(* Logix 5000 project; controller R5_CSS vendor 1 type 14 code 74 rev 19.11; software revision 19.01; part 2 of 20 *)
(* tags used below, declared in another part *)
   AC102A : ANALYTICAL;   // QUENCH WATER CONDUCTIVITY CONTROL
   AlarmMaster : DINT;
   AlarmMasterDisable : BOOL;
   FC101 : FLOW_CONTROL;   // QUENCH BASIN FLOW TRANSMITTER CONTROL
   FC108 : FLOW_CONTROL;   // QUENCH FEED FLOW TRANSMITTER
   FC140A : FLOW_CONTROL;   // QUENCH TOWER UPPER SPRAY FLOW CONTROL
   FC140B : FLOW_CONTROL;   // QUENCH TOWER LOWER SPRAY FLOW CONTROL
   FC215 : FLOW_CONTROL;   // OVERHEAD CONDENSER CHILLED WATER FLOW CONTROL
   FC365 : FLOW_CONTROL;   // COALESCER PROCESS IMPURITY FLOW CONTROL
   FC370 : FLOW_CONTROL;   // COALESCER MAKE UP WATER FLOW CONTROL
   FC403 : FLOW_CONTROL;   // COALESCER FLOW CONTROLLER FEEDS TCV108
   FC406 : FLOW_CONTROL;   // HX COOLING WATER FLOW CONTROL
   LC101 : LEVEL_CONTROL;   // QUENCH TOWER BASIN LIT
   LC205 : LEVEL_CONTROL;   // OVERHEAD CONDENSER BASIN LEVEL CONTROL
   LC302 : LEVEL_CONTROL;   // COALESCER OIL CHAMBER LEVEL CONTROL
   LC304 : LEVEL_CONTROL;   // SETTLER SECONDARY TANK INTERFACE LEVEL
   Major : DINT;
   Minor : DINT;
   My_Gateway : DINT[4];
   My_IP_Address : DINT[4];
   My_Subnet : DINT[4];
   MyDint : DINT;
   P101A : PUMP_CONTROL;
   P101B : PUMP_CONTROL;
   P302A : PUMP_CONTROL;
   P303A : PUMP_CONTROL;
   P303B : PUMP_CONTROL;
   PC101A : PRESSURE_CONTROL;   // LOWER QUENCH TOWER PRESSURE TRANSMITTER
   PC101B : PRESSURE_CONTROL;   // UPPER QUENCH TOWER PRESSURE TRANSMITTER PRESSURE CONTOL
   PC102A : PRESSURE_CONTROL;   // QUENCH BASIN TRANSFER PUMP SUCTION PRESSURE CONTROL
   PC102B : PRESSURE_CONTROL;   // QUENCH BASIN TRANSFER PUMP DISCHARGE PRESSURE CONTROL
   PC132 : PRESSURE_CONTROL;
   PC133 : PRESSURE_CONTROL;
   PC134 : PRESSURE_CONTROL;
   PC214 : PRESSURE_CONTROL;   // VACUUM SYSTEM PRESSURE TRANSMITTER
   PC271 : PRESSURE_CONTROL;   // VENT HEADER PRESSURE CONTROL
   PC407A : PRESSURE_CONTROL;   // PRE HX LOW PRESSURE TRANSMITTER
   PC407B : PRESSURE_CONTROL;   // POST HX LOW PRESSURE TRANSMITTER
   PC408 : PRESSURE_CONTROL;

   PID_JHE102_TON : TIMER := (PRE := 500, ACC := 144, EN := 1, TT := 1);
   PID_JHE114B : PID := (CTL := 4864, OLH := 1, DVPA := 1, PVLA := 1, SP := 130.0, KP := 10.0, KI := 5.0, MAXS := 4095.0, SO := 50.0, MAXO := 50.0, UPD := 1.0, PV := -75.0, ERR := 205.0, OUT := 50.0, MAXI := 4095.0, MAXCV := 100.0, MAXTIE := 4095.0, DATA[0] := 0.009664765, DATA[1] := 29.30403, DATA[2] := -75.0, DATA[3] := 205.0, DATA[4] := 130.0, DATA[5] := 0.024420025, DATA[6] := 1.0, DATA[7] := 16.0, DATA[8] := 10.0, DATA[9] := 5.0, DATA[11] := 10.0, DATA[12] := 5.0, DATA[15] := 1.0, DATA[16] := 0.024420025);
   PID_JHE114B_TON : TIMER := (PRE := 500);
   PID_JHE313A : PID := (CTL := 4231808, NDF := 1, INI := 1, OLH := 1, DVPA := 1, PVHA := 1, SP := 135.0, KP := 10.0, KI := 5.0, MAXS := 200.0, SO := 50.0, MAXO := 50.0, UPD := 1.0, PV := 59.625, ERR := 75.375, OUT := 50.0, MAXI := 200.0, MAXCV := 100.0, MAXTIE := 4095.0, DATA[0] := -484.5469, DATA[1] := -477.0, DATA[2] := 59.625, DATA[3] := 75.375, DATA[4] := 135.0, DATA[5] := 0.5, DATA[6] := 1.0, DATA[7] := 16.0, DATA[8] := 10.0, DATA[9] := 5.0, DATA[11] := 10.0, DATA[12] := 5.0, DATA[15] := 1.0, DATA[16] := 0.024420025);
   PID_JHE313A_TON : TIMER := (PRE := 500, ACC := 16, EN := 1, TT := 1);
   PID_JHE319 : PID := (CTL := 67142400, SWM := 1, INI := 1, DVPA := 1, PVLA := 1, SP := 100.0, KP := 1.0, KI := 1.0, MAXS := 4095.0, MAXO := 50.0, UPD := 1.0, PV := -14.999996, ERR := 115.0, MAXI := 4095.0, MAXCV := 100.0, MAXTIE := 4095.0, DATA[0] := -2.8083029, DATA[1] := 5.8608046, DATA[2] := -14.999996, DATA[3] := 115.0, DATA[4] := 100.0, DATA[5] := 0.024420025, DATA[6] := 1.0, DATA[7] := 16.0, DATA[8] := 1.0, DATA[9] := 1.0, DATA[11] := 1.0, DATA[12] := 1.0, DATA[15] := 1.0, DATA[16] := 0.024420025);   // TEMPERATURE CONTROL OUPUT FOR JHE313B PID
   PID_JHE319_TON : TIMER := (PRE := 500, EN := 1, TT := 1);
   PID_LC370_Enable : BOOL;
   PID_LC370_Enable_ONS : BOOL := 1;
   PID_LC370_Enable_Ton : TIMER := (PRE := 30000);
   PID_LCV370 : PID := (CTL := 71336704, SWM := 1, NDF := 1, INI := 1, DVPA := 1, PVLA := 1, SP := 3.0, KP := 100.0, KI := 200.0, MAXS := 4095.0, SO := 50.0, MAXO := 80.0, UPD := 0.01, PV := -0.00093758106, ERR := 3.0009375, OUT := 50.0, MAXI := 4095.0, MAXCV := 100.0, MAXTIE := 4095.0, DATA[0] := 42.671703, DATA[1] := 0.00036633204, DATA[2] := -0.00093758106, DATA[3] := 3.0009375, DATA[4] := 3.0, DATA[5] := 0.024420025, DATA[6] := 1.0, DATA[7] := 0.16, DATA[8] := 100.0, DATA[9] := 200.0, DATA[11] := 100.0, DATA[12] := 200.0, DATA[15] := 1.0, DATA[16] := 0.024420025);
   PID_LCV370_TON : TIMER := (PRE := 10, EN := 1, TT := 1);
   PID_TC215 : PID := (CTL := 37504, INI := 1, OLH := 1, DVPA := 1, PVHA := 1, SP := 200.0, KP := 0.1, KI := 0.1, MAXS := 4095.0, SO := 100.0, MAXO := 100.0, MINO := 30.0, UPD := 1.0, PV := 59.68126, ERR := 140.31874, OUT := 100.0, MAXI := 4095.0, MAXTIE := 4095.0, DATA[0] := inf, DATA[1] := -23.318686, DATA[2] := 59.68126, DATA[3] := 140.31874, DATA[4] := 200.0, DATA[5] := 0.024420025, DATA[6] := 1.0, DATA[7] := 16.0, DATA[8] := 0.1, DATA[9] := 0.1, DATA[11] := 0.1, DATA[12] := 0.1, DATA[16] := 0.024420025);
   PID_TC215_1 : PID := (CTL := 37376, INI := 1, OLH := 1, DVPA := 1, SP := 100.0, KP := 100.0, KI := 10.0, MAXS := 100.0, MINS := -100.0, SO := 100.0, MAXO := 100.0, MINO := 30.0, UPD := 0.1, PV := 59.49376, ERR := 40.50624, OUT := 100.0, PVH := 100.0, PVL := -100.0, MAXI := 100.0, MINI := -100.0, MAXCV := 100.0, MAXTIE := 4095.0, DATA[0] := inf, DATA[1] := -1275.9501, DATA[2] := 59.49376, DATA[3] := 40.50624, DATA[4] := 100.0, DATA[5] := 0.5, DATA[6] := 1.0, DATA[7] := 1.6, DATA[8] := 100.0, DATA[9] := 10.0, DATA[11] := 100.0, DATA[12] := 10.0, DATA[15] := 1.0, DATA[16] := 0.024420025);
   PID_TC215_TON : TIMER := (PRE := 100, ACC := 47, EN := 1, TT := 1);
   PID_TCV101 : PID := (CTL := 37790848, CA := 1, NDF := 1, INI := 1, OLL := 1, DVNA := 1, PVHA := 1, SP := 15.0, KP := 400.0, KI := 100.0, MAXS := 100.0, DB := 1.0, SO := 5.0, MAXO := 100.0, MINO := 5.0, UPD := 0.1, PV := 13.851999, ERR := -1.1480007, OUT := 5.0, MAXI := 100.0, MAXCV := 100.0, MAXTIE := 4095.0, DATA[0] := 99.62073, DATA[1] := 221.63199, DATA[2] := 13.851999, DATA[3] := -1.1480007, DATA[4] := 15.0, DATA[5] := 1.0, DATA[6] := 1.0, DATA[7] := 1.6, DATA[8] := 400.0, DATA[9] := 100.0, DATA[11] := 400.0, DATA[12] := 100.0, DATA[15] := 1.0, DATA[16] := 0.024420025);
   PID_TCV101_TON : TIMER := (PRE := 100);
   PID_TCV108 : PID := (CTL := 104858880, SWM := 1, CA := 1, NDF := 1, DVNA := 1, PVLA := 1, SP := 145.0, KP := 0.01, KI := 0.05, MAXS := 200.0, SO := 50.0, MAXO := 100.0, MINO := 20.0, UPD := 0.5, PV := -14.999996, ERR := -160.0, OUT := 50.0, MAXI := 200.0, MAXCV := 100.0, MAXTIE := 4095.0, DATA[0] := 50.8, DATA[1] := -119.99997, DATA[2] := -14.999996, DATA[3] := -160.0, DATA[4] := 145.0, DATA[5] := 0.5, DATA[6] := 1.0, DATA[7] := 8.0, DATA[8] := 0.01, DATA[9] := 0.05, DATA[11] := 0.01, DATA[12] := 0.05, DATA[15] := 1.0, DATA[16] := 0.024420025);   // QUENCH FEED CONTROL VALVE
   PID_TCV108_Flow : PID := (CTL := 67142272, SWM := 1, INI := 1, DVPA := 1, PVHA := 1, SP := 75.0, KP := 2.0, KI := 0.5, MAXS := 4095.0, SO := 50.0, MAXO := 100.0, MINO := 20.0, UPD := 0.1, PV := 1.5999985, ERR := 73.4, OUT := 50.0, MAXI := 4095.0, MAXTIE := 4095.0, DATA[0] := 46.415142, DATA[1] := -0.62515205, DATA[2] := 1.5999985, DATA[3] := 73.4, DATA[4] := 75.0, DATA[5] := 0.024420025, DATA[6] := 1.0, DATA[7] := 1.6, DATA[8] := 2.0, DATA[9] := 0.5, DATA[11] := 2.0, DATA[12] := 0.5, DATA[16] := 0.024420025);
   PID_TCV108_TON : TIMER := (PRE := 500, ACC := 297, EN := 1, TT := 1);
   PID_TCV406 : PID := (CTL := 33596544, CA := 1, INI := 1, OLL := 1, DVNA := 1, PVHA := 1, SP := 140.0, KP := 10.0, KI := 1.0, MAXS := 4095.0, SO := 20.0, MAXO := 100.0, MINO := 20.0, UPD := 0.1, PV := 66.33751, ERR := -73.66249, OUT := 20.0, MAXI := 4095.0, MAXCV := 100.0, MAXTIE := 4095.0, DATA[0] := 37.970585, DATA[1] := 25.919418, DATA[2] := 66.33751, DATA[3] := -73.66249, DATA[4] := 140.0, DATA[5] := 0.024420025, DATA[6] := 1.0, DATA[7] := 1.6, DATA[8] := 10.0, DATA[9] := 1.0, DATA[11] := 10.0, DATA[12] := 1.0, DATA[15] := 1.0, DATA[16] := 0.024420025);
   PID_TCV406_TON : TIMER := (PRE := 100, ACC := 109, EN := 1, DN := 1);
   PIT101A_SCP : SCLP := (Input := 9078.0, InputMin := 4000.0, InputMax := 20000.0, ScaledMin := -60.0, ScaledMax := 160.0, Output := 9.822502);   // LOWER QUENCH TOWER PRESSURE TRANSMITTER SCALER
   PIT101B_SCP : SCLP := (Input := 20485.0, InputMin := 4000.0, InputMax := 20000.0, ScaledMin := -60.0, ScaledMax := 160.0, Output := 166.66876);   // UPPER QUENCH TOWER PRESSURE TRANSMITTER SCALER
   PIT102A_SCP : SCLP := (Input := 11045.0, InputMin := 4000.0, InputMax := 20000.0, ScaledMin := -60.0, ScaledMax := 166.0, Output := 39.51062);   // QUENCH BASIN TRANSFER PUMP SUCTION PRESSURE INDICATOR SCALER
   PIT102B_SCP : SCLP := (Input := 4373.0, InputMin := 4000.0, InputMax := 20000.0, ScaledMax := 60.0, Output := 1.3987503);   // QUENCH BASIN TRANSFER PUMP DISCHARGE PRESSURE SCALER
   PIT407A_SCP : SCLP := (Input := 3997.0, InputMin := 4000.0, InputMax := 20000.0, ScaledMax := 100.0, Output := -0.018749237);   // PRE HX LOW PRESSURE TRANSMITTER
   PIT407B_SCP : SCLP := (Input := 3997.0, InputMin := 4000.0, InputMax := 20000.0, ScaledMax := 100.0, Output := -0.018749237);   // POST HX LOW PRESSURE TRANSMITTER SCALER
   PRU_Batch_Start : BOOL[32];
   PRU_Batch_Stop : BOOL[32];
   PRU_BatchNewID : DINT[10] := ([1] := 145, [3] := 148, [4] := 158, [6] := 146, [8] := 161);
   PRU_BLOWER_SEQ : INT;   // PRU BLOWER SEQUENCE NUMBER
   PRU_COOL_REQ : INT;
   PRU_DELAY_REQ : INT;
   PRU_ECOOL_REQ : INT;
   PRU_HOLD_REQ : INT;
   PRU_IDLE_REQ : INT;
   PRU_MaxTempDelayMin : REAL := 45.0;
   PRU_MaxTempDelta : REAL := 50.0;
   PRU_MSG_CommsPath : MSG_CommsPath[9] := ([0].Prefix := '$01$01$12$0E192.168.50.', [0].NodeNum := 106, [0].NodeStr := '106', [0].Path := '$01$01$12$0E192.168.50.106', [1].Prefix := '$01$01$12$0E192.168.50.', [1].NodeNum := 110, [1].NodeStr := '110', [1].Path := '$01$01$12$0E192.168.50.110', [2].Prefix := '$01$01$12$0E192.168.50.', [2].NodeNum := 114, [2].NodeStr := '114', [2].Path := '$01$01$12$0E192.168.50.114', [3].Prefix := '$01$01$12$0E192.168.50.', [3].NodeNum := 118, [3].NodeStr := '118', [3].Path := '$01$01$12$0E192.168.50.118', [4].Prefix := '$01$01$12$0E192.168.50.', [4].NodeNum := 122, [4].NodeStr := '122', [4].Path := '$01$01$12$0E192.168.50.122', [5].Prefix := '$01$01$12$0E192.168.50.', [5].NodeNum := 126, [5].NodeStr := '126', [5].Path := '$01$01$12$0E192.168.50.126', [6].Prefix := '$01$01$12$0E192.168.50.', [6].NodeNum := 130, [6].NodeStr := '130', [6].Path := '$01$01$12$0E192.168.50.130', [7].Prefix := '$01$01$12$0E192.168.50.', [7].NodeNum := 134, [7].NodeStr := '134', [7].Path := '$01$01$12$0E192.168.50.134');
   PRU_MSG_Prefix : STRING := '$01$01$12$0E192.168.50.';
   PRU_PT404 : REAL[10] := ([1] := 538.5, [2] := 540.4, [3] := 532.8, [4] := 586.9, [5] := 516.9, [6] := 379.4, [7] := 572.6, [8] := 744.5);
   PRU_PT404_Done : REAL[10] := ([1] := 722.8, [2] := 697.6, [3] := 709.1, [4] := 717.1, [5] := 697.8, [6] := 699.6, [7] := 711.0, [8] := 698.0);
   PRU_PT404_Max : REAL[10] := ([1] := 772.8, [2] := 747.6, [3] := 759.1, [4] := 767.1, [5] := 747.8, [6] := 749.6, [7] := 761.0, [8] := 748.0);
   PRU_Quantity : DINT := 1;
   PRU_RECIPE_LOAD : INT;
        .0   // PRU A LOAD RECIPE REQUEST
        .1   // PRU B LOAD RECIPE REQUEST
        .2   // PRU C LOAD RECIPE REQUEST
        .3   // PRU D LOAD RECIPE REQUEST
   PRU_RECIPE_LOAD_DLY : TIMER[10] := ([0].PRE := 10000, [1].PRE := 10000, [2].PRE := 10000, [3].PRE := 10000, [4].PRE := 10000, [5].PRE := 10000, [6].PRE := 10000, [7].PRE := 10000);
   PRU_RUNDISABLE : DINT;   // PRU RUN DISABLE
   PRU_RunDoneTemp : BOOL[32];
   PRU_RunDoneTime : BOOL[32];
   PRU_Running : BOOL[32];
   PRU_RunningMaxHrs : REAL := 3.5;
   PRU_RunningMaxMin : REAL;
   PRU_RunningMaxTempDelay : TIMER[10] := ([1].PRE := 2700000, [2].PRE := 2700000, [3].PRE := 2700000, [4].PRE := 2700000, [5].PRE := 2700000, [6].PRE := 2700000, [7].PRE := 2700000, [8].PRE := 2700000);
   PRU_RunningMinutePulse : TIMER[10] := ([1].PRE := 60000, [2].PRE := 60000, [3].PRE := 60000, [4].PRE := 60000, [5].PRE := 60000, [6].PRE := 60000, [7].PRE := 60000, [8].PRE := 60000);
   PRU_RunningTotalMin : COUNTER[10] := ([1].PRE := 210, [2].PRE := 210, [3].PRE := 210, [4].PRE := 210, [5].PRE := 210, [6].PRE := 210, [7].PRE := 210, [8].PRE := 210);
   PRU_SEQ_TMR : TIMER := (PRE := 1000);   // PRU_SEQUENCE TIMER
   PRU_START_REQ : INT;
        .0   // PRU A Start Request
   PRU_STARTDISABLE : DINT;   // PRU START DISABLE
        .0   // P101A/P101B START DISABLE
        .1   // P302A/B START DISABLE
   PRU_TT303 : REAL[10] := ([1] := 50.5, [2] := 50.0, [3] := 51.5, [4] := 51.3, [5] := 50.1, [6] := 50.3, [7] := 51.4, [8] := 51.4);
   PRU_TT404 : REAL[10] := ([1] := 51.7, [2] := 52.6, [3] := 52.5, [4] := 52.0, [5] := 52.6, [6] := 53.7, [7] := 52.4, [8] := 51.8);
   PRUA_Batch_Start_ONS : BOOL;
   PRUA_Batch_Stop_ONS : BOOL := 1;
   PRUA_CHANGE : INT := 4;
   PRUA_CHANGE_OF_STATE : BOOL := 1;
   PRUA_COMMS_TIMER : TIMER := (PRE := 60000, ACC := 60009, EN := 1, DN := 1);
   PRUA_ECOOL : BOOL;
   PRUA_ECOOL_TON : TIMER := (PRE := 5000);
   PRUA_ERR_MSG_OUTPUT : BOOL;
   PRUA_HeartbeatCommsLoss : BOOL := 1;
   PRUA_HeartbeatOffONS : BOOL := 1;
   PRUA_HeartbeatOnONS : BOOL;
   PRUA_HeartbeatToggle : BOOL;
   PRUA_MSG_ALM : AlarmAOI := (Type := 3);
   PRUA_MSG_ERROR : COUNTER := (ACC := 2, CU := 1, DN := 1);
   PRUA_MSG_STORAGE : BOOL := 1;
   PRUA_READ : INT[30] := ([0] := -32768, [1] := 22656, [2] := 21, [3] := 64, [4] := 28960, [5] := 392, [6] := 2, [7] := 75, [10] := 501, [11] := 498, [12] := 1000, [13] := 12, [14] := 1000, [15] := 1000, [16] := 15, [17] := 505, [18] := 1076, [19] := 517, [20] := 1, [23] := 359, [24] := 31);
        [0].3   // Temper Mode (temper=1)
        [1].3   // Combustion Blower Start Request
        [1].4   // PRU COMBUSTION BURNER ALARM
        [1].5   // Pru Combustion Burner Limits Complete Bit
        [1].6   // Combustion Burner Purge Status
        [1].7   // Combustion Burner Low Fire Command
        [1].8   // Combustion Burnrer Ignition Status
        [1].9   // Combustion Burner Main Burner On
        [1].10   // Burner Release to Auto
        [1].11   // Combustion Burner Auto Status
        [1].12   // Combustion Blower Auto Status
        [1].14   // Fresh Air Damper Open Switch
        [2]   // DCC VAC PRESSURE
        [1].15   // Fresh Air Damper Closed Switch
        [3].0   // PRU START VISIBLE TO HMI
        [3].1   // IDLE PUSH BUTTON VISIBLE
        [3].2   // COOL VISIBLE
        [3].3   // PRU OK TO SWAP/OPEN
        [3].4   // TEMPER PB VISIBLE
        [6]   // Burner status 0=off, 1= man on, 2 = auto off, 3 = auto on
        [8]   // Exhaust Damper % open x 10
        [9]   // Fresh Air Damper % open
        [10]   // TIC201
        [11]   // TIC202
        [16]   // PIC401
        [17]   // TIC303
        [18]   // TIC330_OP
        [19]   // TIC404
        [20].0   // PRU IN ECOOL
        [0].0   // PRU heart beat
        [0].14   // Burner Released to Auto (Started)
        [0].15   // Stop signal from either new start or low temperature
        [0].1   // local remote push button (local=1)
   PRUA_READ_MSG : MESSAGE;
        MessageParameters(ServiceCode := 16#0fa2, LocalElement := PRUA_READ[0], ...)
   PRUA_READ_MSG_ER_Count : COUNTER := (PRE := 9999);
   PRUA_READ_MSG_ER_ONS1 : BOOL := 1;
   PRUA_START_REQ_ONS : BOOL[32];
   PRUA_WERR_MSG_OUTPUT : BOOL;
   PRUA_WMSG_ERROR : COUNTER;
   PRUA_WMSG_STORAGE : BOOL;
   PRUA_WRITE : INT[40] := ([0] := 96, [3] := 4, [4] := 60, [12] := 825, [13] := 950, [14] := 1100, [15] := 1000, [22] := 30, [23] := 10, [24] := 7, [32] := 600, [33] := 900, [34] := 1500);
        [0]   // CMD WORD TO PRU
        [0].0   // CMD WORD TO PRU CSS HEARTBEAT
        [0].2   // CMD WORD TO PRU LOAD RECIPE
        [0].6   // CMD WORD TO PRU FACILTY PWR ON 1=OK
        [0].3   // CMD WORD TO PRU DELAY START REQUEST 1=REQ
        [0].1   // CMD WORD TO PRU OK TO RUN "PRU_RUN_DISABLE" 1=OK
        [0].4   // CMD WORD TO PRU GEN POWER ON SEQUENCED START 1=START BLOWER
        [0].5   // CMD WORD TO PRU OK TO START "PRU_START_DISABLE" 1=OK
        [0].7   // CMD WORD TO PRU TEST MODE ENABLED 1=ENABLED
   PRUA_WRITE_MSG : MESSAGE;
        MessageParameters(ServiceCode := 16#0faa, LocalElement := PRUA_WRITE[0], ...)
   PRUA_WRITE_MSG_ER_Count : COUNTER := (PRE := 9999);
   PRUA_WRITE_MSG_ER_ONS1 : BOOL := 1;
   PRUB_Batch_Start_ONS : BOOL;
   PRUB_Batch_Stop_ONS : BOOL := 1;
   PRUB_CHANGE : INT := 5;
   PRUB_CHANGE_OF_STATE : BOOL := 1;
   PRUB_COMMS_TIMER : TIMER := (PRE := 60000, ACC := 60009, EN := 1, DN := 1);
   PRUB_ECOOL : BOOL;
   PRUB_ECOOL_TON : TIMER := (PRE := 5000);
   PRUB_ERR_MSG_OUTPUT : BOOL;
   PRUB_HeartbeatCommsLoss : BOOL := 1;
   PRUB_HeartbeatOffONS : BOOL;
   PRUB_HeartbeatOnONS : BOOL := 1;
   PRUB_HeartbeatToggle : BOOL;
   PRUB_MSG_ERROR : COUNTER := (ACC := 56, CU := 1, DN := 1);
   PRUB_MSG_STORAGE : BOOL := 1;
   PRUB_READ : INT[30] := ([0] := -32767, [1] := -26496, [2] := 20, [3] := 69, [4] := 28960, [5] := 392, [6] := 2, [7] := 65, [9] := -1, [10] := 504, [11] := 493, [12] := 1000, [13] := 12, [15] := 1000, [16] := 6, [17] := 500, [18] := 1073, [19] := 526, [23] := 468, [24] := 38);
        [0].0   // HEARTBEAT BIT FROM PRU
        [14]   // FRESH AIR AUTOMATIC SETPOINT
        [15]   // FRESH AIR MANUAL SETPOINT
        [20].0   // PRU IN ECOOL
        [0].1   // local remote push button (local=1)
        [0].3   // Temper Mode (temper=1)
   PRUB_READ_MSG : MESSAGE;
        MessageParameters(ServiceCode := 16#0fa2, LocalElement := PRUB_READ[0], ...)
   PRUB_RECIPE_LOAD : INT;
        .0   // PRU A LOAD RECIPE REQUEST
        .1   // PRU B LOAD RECIPE REQUEST
        .2   // PRU C LOAD RECIPE REQUEST
        .3   // PRU D LOAD RECIPE REQUEST
   PRUB_START_REQ_ONS : BOOL[32];
   PRUB_TEMP : INT;   // TEST
   PRUB_WERR_MSG_OUTPUT : BOOL;
   PRUB_WMSG_ERROR : COUNTER := (ACC := 55, CU := 1, DN := 1);
   PRUB_WMSG_STORAGE : BOOL := 1;
   PRUB_WRITE : INT[40] := ([0] := 97, [3] := 5, [4] := 60, [12] := 825, [13] := 950, [14] := 1100, [15] := 1000, [22] := 30, [23] := 10, [24] := 7, [32] := 600, [33] := 900, [34] := 1500);
        [0].3   // CMD WORD TO PRU DELAY START REQUEST 1=REQ
        [0]   // CMD WORD TO PRU
        [0].0   // CMD WORD TO PRU CSS HEARTBEAT
        [0].2   // CMD WORD TO PRU LOAD RECIPE
        [0].1   // CMD WORD TO PRU OK TO RUN "PRU_RUN_DISABLE" 1=OK
        [0].5   // CMD WORD TO PRU OK TO START "PRU_START_DISABLE" 1=OK
        [0].6   // CMD WORD TO PRU FACILTY PWR ON 1=OK
        [0].4   // CMD WORD TO PRU GEN POWER ON SEQUENCED START 1=START BLOWER
        [0].7   // CMD WORD TO PRU TEST MODE ENABLED 1=ENABLED
   PRUB_WRITE_MSG : MESSAGE;
        MessageParameters(ServiceCode := 16#0faa, LocalElement := PRUB_WRITE[0], ...)
   PRUC_Batch_Start_ONS : BOOL;
   PRUC_Batch_Stop_ONS : BOOL := 1;
   PRUC_CHANGE : INT := 1;
   PRUC_CHANGE_OF_STATE : BOOL := 1;
   PRUC_COMMS_TIMER : TIMER := (PRE := 60000, ACC := 60009, EN := 1, DN := 1);
   PRUC_ECOOL : BOOL;
   PRUC_ECOOL_TON : TIMER := (PRE := 5000);
   PRUC_HeartbeatCommsLoss : BOOL := 1;
   PRUC_HeartbeatOffONS : BOOL;
   PRUC_HeartbeatOnONS : BOOL := 1;
   PRUC_HeartbeatToggle : BOOL;
   PRUC_READ : INT[30] := ([0] := -32767, [1] := 22656, [2] := 21, [3] := 64, [4] := 28960, [5] := 456, [6] := 2, [7] := 75, [10] := 513, [11] := 505, [12] := 1000, [13] := 12, [14] := 1000, [15] := 1000, [16] := -10, [17] := 515, [18] := 1057, [19] := 525, [20] := 1, [23] := 359, [24] := 44);
        [20].0   // PRU IN ECOOL
        [0].3   // Temper Mode (temper=1)
        [0].1   // local remote push button (local=1)
   PRUC_READ_MSG : MESSAGE;
        MessageParameters(ServiceCode := 16#0fa2, LocalElement := PRUC_READ[0], ...)
   PRUC_RECIPE_LOAD : INT;
        .0   // PRU A LOAD RECIPE REQUEST
        .1   // PRU B LOAD RECIPE REQUEST
        .2   // PRU C LOAD RECIPE REQUEST
        .3   // PRU D LOAD RECIPE REQUEST
   PRUC_START_REQ_ONS : BOOL[32];
   PRUC_WRITE : INT[40] := ([0] := 96, [3] := 1, [4] := 60, [12] := 825, [13] := 950, [14] := 1100, [15] := 1000, [22] := 30, [23] := 10, [24] := 7, [32] := 600, [33] := 900, [34] := 1500);
        [0]   // CMD WORD TO PRU
        [0].2   // CMD WORD TO PRU LOAD RECIPE
        [0].0   // CMD WORD TO PRU CSS HEARTBEAT
        [0].1   // CMD WORD TO PRU OK TO RUN "PRU_RUN_DISABLE" 1=OK
        [0].3   // CMD WORD TO PRU DELAY START REQUEST 1=REQ
        [0].4   // CMD WORD TO PRU GEN POWER ON SEQUENCED START 1=START BLOWER
        [0].5   // CMD WORD TO PRU OK TO START "PRU_START_DISABLE" 1=OK
        [0].6   // CMD WORD TO PRU FACILTY PWR ON 1=OK
        [0].7   // CMD WORD TO PRU TEST MODE ENABLED 1=ENABLED
   PRUC_WRITE_MSG : MESSAGE;
        MessageParameters(ServiceCode := 16#0faa, LocalElement := PRUC_WRITE[0], ...)
   PRUD_Batch_Start_ONS : BOOL;
   PRUD_Batch_Stop_ONS : BOOL := 1;
   PRUD_CHANGE : INT := 1;
   PRUD_CHANGE_OF_STATE : BOOL := 1;
   PRUD_COMMS_TIMER : TIMER := (PRE := 60000, ACC := 60009, EN := 1, DN := 1);
   PRUD_ECOOL : BOOL;
   PRUD_ECOOL_TON : TIMER := (PRE := 5000);
   PRUD_HeartbeatCommsLoss : BOOL := 1;
   PRUD_HeartbeatOffONS : BOOL := 1;
   PRUD_HeartbeatOnONS : BOOL;
   PRUD_HeartbeatToggle : BOOL;
   PRUD_READ : INT[30] := ([0] := -32768, [1] := 22656, [2] := 21, [3] := 64, [4] := 28960, [5] := 392, [6] := 2, [7] := 75, [8] := -2, [10] := 505, [11] := 514, [12] := 1000, [13] := 12, [14] := 1000, [15] := 1000, [16] := 28, [17] := 513, [18] := 1057, [19] := 520, [20] := 1, [23] := 359, [24] := 29);   // PRU D READ
        [20].0   // PRU IN ECOOL
        [0].1   // local remote push button (local=1)
        [0].3   // Temper Mode (temper=1)
   PRUD_READ_MSG : MESSAGE;
        MessageParameters(ServiceCode := 16#0fa2, LocalElement := PRUD_READ[0], ...)
   PRUD_RECIPE_LOAD : INT;
        .0   // PRU A LOAD RECIPE REQUEST
        .1   // PRU B LOAD RECIPE REQUEST
        .2   // PRU C LOAD RECIPE REQUEST
        .3   // PRU D LOAD RECIPE REQUEST
   PRUD_START_REQ_ONS : BOOL[32];
   PRUD_WRITE : INT[40] := ([0] := 97, [3] := 1, [4] := 60, [12] := 825, [13] := 950, [14] := 1100, [15] := 1000, [22] := 30, [23] := 10, [24] := 7, [32] := 600, [33] := 900, [34] := 1500);
        [0]   // CMD WORD TO PRU
        [0].0   // CMD WORD TO PRU CSS HEARTBEAT
        [0].2   // CMD WORD TO PRU LOAD RECIPE
        [0].1   // CMD WORD TO PRU OK TO RUN "PRU_RUN_DISABLE" 1=OK
        [0].3   // CMD WORD TO PRU DELAY START REQUEST 1=REQ
        [0].4   // CMD WORD TO PRU GEN POWER ON SEQUENCED START 1=START BLOWER
        [0].5   // CMD WORD TO PRU OK TO START "PRU_START_DISABLE" 1=OK
        [0].6   // CMD WORD TO PRU FACILTY PWR ON 1=OK
        [0].7   // CMD WORD TO PRU TEST MODE ENABLED 1=ENABLED
   PRUD_WRITE_MSG : MESSAGE;
        MessageParameters(ServiceCode := 16#0faa, LocalElement := PRUD_WRITE[0], ...)
   PRUE_Batch_Start_ONS : BOOL;
   PRUE_Batch_Stop_ONS : BOOL := 1;
   PRUE_CHANGE : INT := 5;
   PRUE_CHANGE_OF_STATE : BOOL := 1;
   PRUE_COMMS_TIMER : TIMER := (PRE := 60000, ACC := 60005, EN := 1, DN := 1);
   PRUE_ECOOL : BOOL;
   PRUE_ECOOL_TON : TIMER := (PRE := 5000);
   PRUE_ERR_MSG_OUTPUT : BOOL;
   PRUE_HeartbeatCommsLoss : BOOL := 1;
   PRUE_HeartbeatOffONS : BOOL := 1;
   PRUE_HeartbeatOnONS : BOOL;
   PRUE_HeartbeatToggle : BOOL;
   PRUE_MSG_ALM : AlarmAOI;
   PRUE_MSG_ERROR : COUNTER;
   PRUE_MSG_STORAGE : BOOL;
   PRUE_READ : INT[30] := ([0] := -32768, [1] := -26496, [2] := 20, [3] := 69, [4] := 28960, [5] := 392, [6] := 2, [7] := 65, [10] := 504, [11] := 503, [12] := 1000, [13] := 12, [15] := 1000, [16] := -15, [17] := 501, [18] := 1070, [19] := 526, [23] := 470, [24] := 23);
   PRUE_READ_MSG : MESSAGE;
        MessageParameters(ServiceCode := 16#0fa2, LocalElement := PRUE_READ[0], ...)
   PRUE_READ_MSG_ER_Count : COUNTER;
   PRUE_READ_MSG_ER_ONS1 : BOOL;
   PRUE_START_REQ_ONS : BOOL[32];
   PRUE_WERR_MSG_OUTPUT : BOOL;
   PRUE_WMSG_ERROR : COUNTER;
   PRUE_WMSG_STORAGE : BOOL;
   PRUE_WRITE : INT[40] := ([0] := 96, [3] := 5, [4] := 60, [12] := 825, [13] := 950, [14] := 1100, [15] := 1000, [22] := 30, [23] := 10, [24] := 7, [32] := 600, [33] := 900, [34] := 1500);
   PRUE_WRITE_MSG : MESSAGE;
        MessageParameters(ServiceCode := 16#0faa, LocalElement := PRUE_WRITE[0], ...)
   PRUE_WRITE_MSG_ER_Count : COUNTER;
   PRUE_WRITE_MSG_ER_ONS1 : BOOL;
   PRUF_Batch_Start_ONS : BOOL;
   PRUF_Batch_Stop_ONS : BOOL := 1;
   PRUF_CHANGE : INT := 5;
   PRUF_CHANGE_OF_STATE : BOOL := 1;
   PRUF_COMMS_TIMER : TIMER := (PRE := 60000, ACC := 60005, EN := 1, DN := 1);
   PRUF_ECOOL : BOOL;
   PRUF_ECOOL_TON : TIMER := (PRE := 5000);
   PRUF_ERR_MSG_OUTPUT : BOOL;
   PRUF_HeartbeatCommsLoss : BOOL := 1;
   PRUF_HeartbeatOffONS : BOOL;
   PRUF_HeartbeatOnONS : BOOL := 1;
   PRUF_HeartbeatToggle : BOOL;
   PRUF_MSG_ALM : AlarmAOI;
   PRUF_MSG_ERROR : COUNTER;
   PRUF_MSG_STORAGE : BOOL;
   PRUF_READ : INT[30] := ([0] := -32767, [1] := -26624, [2] := 52, [3] := 69, [4] := 28960, [5] := 392, [6] := 2, [7] := 65, [10] := 512, [11] := 506, [12] := 1000, [13] := 12, [15] := 1000, [16] := -20, [17] := 503, [18] := 1064, [19] := 537, [23] := 456, [24] := 42);
   PRUF_READ_MSG : MESSAGE;
        MessageParameters(ServiceCode := 16#0fa2, LocalElement := PRUF_READ[0], ...)
   PRUF_READ_MSG_ER_Count : COUNTER;
   PRUF_READ_MSG_ER_ONS1 : BOOL;
   PRUF_START_REQ_ONS : BOOL[32];
   PRUF_WERR_MSG_OUTPUT : BOOL;
   PRUF_WMSG_ERROR : COUNTER;
   PRUF_WMSG_STORAGE : BOOL;
   PRUF_WRITE : INT[40] := ([0] := 96, [3] := 5, [4] := 60, [12] := 825, [13] := 950, [14] := 1100, [15] := 1000, [22] := 30, [23] := 10, [24] := 7, [32] := 600, [33] := 900, [34] := 1500);
   PRUF_WRITE_MSG : MESSAGE;
        MessageParameters(ServiceCode := 16#0faa, LocalElement := PRUF_WRITE[0], ...)
   PRUF_WRITE_MSG_ER_Count : COUNTER;
   PRUF_WRITE_MSG_ER_ONS1 : BOOL;
   PRUG_Batch_Start_ONS : BOOL;
   PRUG_Batch_Stop_ONS : BOOL := 1;
   PRUG_CHANGE : INT := 5;
   PRUG_CHANGE_OF_STATE : BOOL;
   PRUG_COMMS_TIMER : TIMER := (PRE := 60000, ACC := 60005, EN := 1, DN := 1);
   PRUG_ECOOL : BOOL;
   PRUG_ECOOL_TON : TIMER := (PRE := 5000);
   PRUG_ERR_MSG_OUTPUT : BOOL;
   PRUG_HeartbeatCommsLoss : BOOL := 1;
   PRUG_HeartbeatOffONS : BOOL;
   PRUG_HeartbeatOnONS : BOOL := 1;
   PRUG_HeartbeatToggle : BOOL;
   PRUG_MSG_ALM : AlarmAOI;
   PRUG_MSG_ERROR : COUNTER;
   PRUG_MSG_STORAGE : BOOL;
   PRUG_READ : INT[30] := ([0] := -32767, [1] := -26496, [2] := 20, [3] := 69, [4] := 28960, [5] := 392, [6] := 2, [7] := 65, [9] := -1, [10] := 504, [11] := 462, [12] := 1000, [13] := 12, [15] := 1000, [16] := -11, [17] := 514, [18] := 1060, [19] := 524, [23] := 451, [24] := 55);
   PRUG_READ_MSG : MESSAGE;
        MessageParameters(ServiceCode := 16#0fa2, LocalElement := PRUG_READ[0], ...)
   PRUG_READ_MSG_ER_Count : COUNTER;
   PRUG_READ_MSG_ER_ONS1 : BOOL;
   PRUG_START_REQ_ONS : BOOL[32];
   PRUG_WERR_MSG_OUTPUT : BOOL;
   PRUG_WMSG_ERROR : COUNTER;
   PRUG_WMSG_STORAGE : BOOL;
   PRUG_WRITE : INT[40] := ([0] := 96, [3] := 5, [4] := 60, [12] := 825, [13] := 950, [14] := 1100, [15] := 1000, [22] := 30, [23] := 10, [24] := 7, [32] := 600, [33] := 900, [34] := 1500);
   PRUG_WRITE_MSG : MESSAGE;
        MessageParameters(ServiceCode := 16#0faa, LocalElement := PRUG_WRITE[0], ...)
   PRUG_WRITE_MSG_ER_Count : COUNTER;
   PRUG_WRITE_MSG_ER_ONS1 : BOOL;
   PRUH_Batch_Start_ONS : BOOL;
   PRUH_Batch_Stop_ONS : BOOL := 1;
   PRUH_CHANGE : INT := 4;
   PRUH_CHANGE_OF_STATE : BOOL := 1;
   PRUH_COMMS_TIMER : TIMER := (PRE := 60000, ACC := 60005, EN := 1, DN := 1);
   PRUH_ECOOL : BOOL;
   PRUH_ECOOL_TON : TIMER := (PRE := 5000);
   PRUH_ERR_MSG_OUTPUT : BOOL;
   PRUH_HeartbeatCommsLoss : BOOL := 1;
   PRUH_HeartbeatOffONS : BOOL;
   PRUH_HeartbeatOnONS : BOOL := 1;
   PRUH_HeartbeatToggle : BOOL;
   PRUH_MSG_ALM : AlarmAOI;
   PRUH_MSG_ERROR : COUNTER;
   PRUH_MSG_STORAGE : BOOL;
   PRUH_READ : INT[30] := ([0] := -32767, [1] := -26496, [2] := 20, [3] := 69, [4] := 28960, [5] := 392, [6] := 2, [7] := 65, [8] := -1, [10] := 502, [11] := 496, [12] := 1000, [13] := 12, [15] := 1000, [16] := -24, [17] := 514, [18] := 1100, [19] := 518, [23] := 385, [24] := 2);
   PRUH_READ_MSG : MESSAGE;
        MessageParameters(ServiceCode := 16#0fa2, LocalElement := PRUH_READ[0], ...)
   PRUH_READ_MSG_ER_Count : COUNTER;
   PRUH_READ_MSG_ER_ONS1 : BOOL;
   PRUH_START_REQ_ONS : BOOL[32];
   PRUH_WERR_MSG_OUTPUT : BOOL;
   PRUH_WMSG_ERROR : COUNTER;
   PRUH_WMSG_STORAGE : BOOL;
   PRUH_WRITE : INT[40] := ([0] := 96, [3] := 4, [4] := 60, [12] := 825, [13] := 950, [14] := 1100, [15] := 1000, [22] := 30, [23] := 10, [24] := 7, [32] := 600, [33] := 900, [34] := 1500);
   PRUH_WRITE_MSG : MESSAGE;
        MessageParameters(ServiceCode := 16#0faa, LocalElement := PRUH_WRITE[0], ...)
   PRUH_WRITE_MSG_ER_Count : COUNTER;
   PRUH_WRITE_MSG_ER_ONS1 : BOOL;
   PT271_SCP : SCLP := (Input := 15894.0, InputMin := 4000.0, InputMax := 20000.0, ScaledMin := -10.0, ScaledMax := 10.0, Output := 4.8675003);   // VENT HEADER PRESSURE TRANSMITTER SCALER
   PY214_SCP : SCLP := (Input := 3200.0, InputMin := 4000.0, InputMax := 20000.0, ScaledMax := 100.0, Output := -5.0);
   PY271_SCP : SCLP := (Input := 3200.0, InputMin := 4000.0, InputMax := 20000.0, ScaledMax := 100.0, Output := -5.0);
   QA_JC306 : PUMP_CONTROL;
   QUENCH_TOWER : SCLP;
   QuenchFlowAutoControl : BOOL := 1;
   QuenchFlowAutoControlPB : BOOL;
   QuenchFlowAutoControlPB_ONS : BOOL;
   QuenchFlowMeterFailed : BOOL;
   QuenchFlowMeterFailedONS1 : BOOL;
   QuenchFlowMeterFailedONS2 : BOOL;
   QuenchFlowMeterFailedTOF : TIMER := (PRE := 30000, ACC := 30000);
   QuenchTowerControlMode : BOOL := 1;   // 0 = Temp.control 1 = Flow control
   RandomNumber : REAL := 0.054;
   RandomNumberDint : DINT := 54;
   Revision : DINT := 5;
   SetMyIP_Enabled : BOOL;
   SignalLossHigh_IF8 : DINT := 21000;
   SignalLossLow_IF8 : DINT := 3810;
   SLOT01 : INT;
   SLOT02 : INT;
   SLOT03 : REAL[8];
   SLOT04 : REAL[8];
   SLOT05 : REAL[8];
   SLOT06 : REAL[8];
   SLOT07 : REAL[8];
   SLOT08 : REAL[8];
   SLOT09 : REAL[8];
   SLOT10 : REAL[8];
   SLOT11 : REAL[8];
   SLOT12 : REAL[8];
   SLOT13 : DINT := 1024;
   SpareAI : AnalogControl := (RawCounts := 3200);
   SpareAO_SCLP : SCLP := (InputMax := 100.0, ScaledMin := 4000.0, ScaledMax := 20000.0, Output := 4000.0);
   SpareSimulate : BOOL;
   TAS15569 : BOOL := 1;
   TC101A : TEMP_CONTROL := (FB := 34.576, TT := 63.581253, TALL_SP := 75.0, TAL_SP := 81000.0, TAH_SP := 160.0, TAHH_SP := 180.0, TALL := 1, TAL := 1, TALL_TMR.PRE := 5000, TALL_TMR.ACC := 5009, TALL_TMR.EN := 1, TALL_TMR.DN := 1, TAL_TMR.PRE := 5000, TAL_TMR.ACC := 5009, TAL_TMR.EN := 1, TAL_TMR.DN := 1, TAH_TMR.PRE := 5000, TAHH_TMR.PRE := 5000, TAHH_DEV := 178.0, TAH_DEV := 158.0, TAL_DEV := 81002.0, TALL_DEV := 77.0, RawCounts := 7391);   // QUENCH BASIN TRANSFER BASIN A TEMPERATURE CONTROL
   TC101B : TEMP_CONTROL := (TT := 63.975006, TALL_SP := 95.0, TAL_SP := 105.0, TAH_SP := 160.0, TAHH_SP := 180.0, TALL := 1, TAL := 1, TALL_TMR.PRE := 5000, TALL_TMR.ACC := 5009, TALL_TMR.EN := 1, TALL_TMR.DN := 1, TAL_TMR.PRE := 5000, TAL_TMR.ACC := 5009, TAL_TMR.EN := 1, TAL_TMR.DN := 1, TAH_TMR.PRE := 5000, TAHH_TMR.PRE := 5000, TAHH_DEV := 178.0, TAH_DEV := 158.0, TAL_DEV := 107.0, TALL_DEV := 97.0, RawCounts := 7412);   // QUENCH BASIN TRANSFER BASIN B TEMPERATURE CONTROL
   TC108 : TEMP_CONTROL := (MAN_SP := 50.0, AUTO_SP := 100.0, CO := 50.0, FB := 50.0, TT := 69.5625, TALL_SP := 100.0, TAL_SP := 120.0, TAH_SP := 160.0, TAHH_SP := 170.0, TALL := 1, TAL := 1, TALL_TMR.PRE := 5000, TALL_TMR.ACC := 5008, TALL_TMR.EN := 1, TALL_TMR.DN := 1, TAL_TMR.PRE := 5000, TAL_TMR.ACC := 5008, TAL_TMR.EN := 1, TAL_TMR.DN := 1, TAH_TMR.PRE := 5000, TAHH_TMR.PRE := 5000, TAHH_DEV := 168.0, TAH_DEV := 158.0, TAL_DEV := 122.0, TALL_DEV := 102.0, RawCounts := 7710);   // QUENCH TOWER EXIT GAS TEMPERATURE CONTROL
   TC108_AUTO_ONS1 : BOOL;
   TC108_AUTO_ONS2 : BOOL := 1;
   TC108_AutoStatic_SeekMaxSec : DINT := 120;
   TC108_AutoStatic_SeekMaxTime : BOOL;
   TC108_AutoStatic_SeekMaxTmr : TIMER := (PRE := 120000);
   TC108_AutoStatic_SeekTmr : TIMER := (PRE := 5000);
   TC108_AutoStatic_SP : REAL := 50.0;
   TC108_AutoStatic_SP_DB : REAL := 2.0;
   TC108_AutoStatic_SP_DB_Down : REAL;
   TC108_AutoStatic_SP_DB_Up : REAL;
   TC108_manual_ONS1 : BOOL;
   TC108_QuenchFlowMeterFailedHold : REAL := 40.0;
   TC108_QuenchFlowMeterFailedONS : BOOL;
   TC108_StaticMode : BOOL := 1;
   TC108_StaticMode_Seek : BOOL;
   TC110 : TEMP_CONTROL := (TT := -75.0, TALL_SP := 115.0, TAL_SP := 125.0, TAH_SP := 212.0, TAHH_SP := 250.0, TALL := 1, TAL := 1, TALL_TMR.PRE := 5000, TALL_TMR.ACC := 5005, TALL_TMR.EN := 1, TALL_TMR.DN := 1, TAL_TMR.PRE := 5000, TAL_TMR.ACC := 5005, TAL_TMR.EN := 1, TAL_TMR.DN := 1, TAH_TMR.PRE := 5000, TAHH_TMR.PRE := 5000, TAHH_DEV := 245.0, TAH_DEV := 207.0, TAL_DEV := 130.0, TALL_DEV := 120.0, XA := 1);   // Quench Water Cartridge Heater Bundle Temp
   TC110_SCP : SCLP := (InputMin := 4000.0, InputMax := 20000.0, ScaledMax := 300.0, Output := -75.0);
   TC112 : TEMP_CONTROL := (AUTO_SP := 135.0, TT := 64.05, TALL_SP := 120.0, TAL_SP := 125.0, TAH_SP := 140.0, TAHH_SP := 150.0, TALL := 1, TAL := 1, TALL_TMR.PRE := 5000, TALL_TMR.ACC := 5008, TALL_TMR.EN := 1, TALL_TMR.DN := 1, TAL_TMR.PRE := 5000, TAL_TMR.ACC := 5008, TAL_TMR.EN := 1, TAL_TMR.DN := 1, TAH_TMR.PRE := 5000, TAHH_TMR.PRE := 5000, TAHH_DEV := 145.0, TAH_DEV := 135.0, TAL_DEV := 130.0, TALL_DEV := 125.0, XA := 1, kWh_Tmr.PRE := 1000, kWh_SampleTime := 1.0, kWh_TimeMultiplier := 3600.0);   // Quench Water Cartridge Heater ProcessTemp
   TC112_AUTO_Ons : BOOL;
   TC112_AUTO_Ons1 : BOOL := 1;
   TC112_HeaterDisabled : BOOL := 1;
   TC112_MANUAL_Ons : BOOL := 1;
   TC112_NoPumpsRunningAlm : BOOL;
   TC112_SCP : SCLP := (Input := 7414.0, InputMin := 4000.0, InputMax := 20000.0, ScaledMax := 300.0, Output := 64.01251);
   TC112_START_TON : TIMER := (PRE := 5000);
   TC112A : TEMP_CONTROL := (TALL_TMR.PRE := 5000, TAL_TMR.PRE := 5000, TAH_TMR.PRE := 5000, TAHH_TMR.PRE := 5000, TAHH_DEV := -5.0, TAH_DEV := -5.0, TAL_DEV := 5.0, TALL_DEV := 5.0);
   TC114_HeaterDisabled : BOOL;
   TC114A : TEMP_CONTROL := (MANUAL := 1, TT := 64.20001, TAH_SP := 280.0, TAHH_SP := 300.0, TALL_TMR.PRE := 5000, TAL_TMR.PRE := 5000, TAH_TMR.PRE := 5000, TAHH_TMR.PRE := 5000, TAHH_DEV := 295.0, TAH_DEV := 275.0, TAL_DEV := 5.0, TALL_DEV := 5.0, RUN_STATUS := 1, RawCounts := 7424);   // QUENCH BASIN SHELL TEMPERATURE CONTROL
   TC114B : TEMP_CONTROL := (AUTO := 1, MAN_SP := 50.0, AUTO_SP := 130.0, PID_CO := 50.0, TT := 64.256256, TALL_SP := 90.0, TAL_SP := 100.0, TAH_SP := 150.0, TAHH_SP := 160.0, TALL_TMR.PRE := 5000, TAL_TMR.PRE := 5000, TAH_TMR.PRE := 5000, TAHH_TMR.PRE := 5000, TAHH_DEV := 155.0, TAH_DEV := 145.0, TAL_DEV := 105.0, TALL_DEV := 95.0, RawCounts := 7427);   // QUENCH BASIN LIQUID TEMPERATURE CONTROL
   TC114B_AUTO_Ons : BOOL := 1;
   TC114B_AUTO_Ons1 : BOOL := 1;
   TC114B_MANUAL_Ons : BOOL := 1;
   TC121 : TEMP_CONTROL := (TAH_SP := 900.0, TAHH_SP := 950.0, TDAH_SP := 200.0, TAH_TMR.PRE := 5000, TAHH_TMR.PRE := 5000, TAHH_DEV := 945.0, TAH_DEV := 895.0, TDAH_DEV := 195.0);
   TC121A : TEMP_CONTROL := (TT := -250.0, TAL_SP := 50.0, TAH_SP := 900.0, TAHH_SP := 950.0, TDAH_SP := 100.0, DIFFERENCE := -301.7, TALL_TMR.PRE := 5000, TAL_TMR.PRE := 5000, TAH_TMR.PRE := 5000, TAHH_TMR.PRE := 5000, TDAH_TMR.PRE := 5000, TAHH_DEV := 945.0, TAH_DEV := 895.0, TAL_DEV := 55.0, TALL_DEV := 5.0, TDAH_DEV := 95.0, XA := 1);   // GTL FROM PRUA TEMPERATURE CONTROL
   TC121B : TEMP_CONTROL := (TT := -250.0, TAH_SP := 900.0, TAHH_SP := 950.0, DIFFERENCE := -302.6, TALL_TMR.PRE := 5000, TALL_TMR.ACC := 5000, TAL_TMR.PRE := 5000, TAL_TMR.ACC := 5002, TAH_TMR.PRE := 5000, TAHH_TMR.PRE := 5000, TDAH_TMR.PRE := 5000, TAHH_DEV := 945.0, TAH_DEV := 895.0, TDAH_DEV := -5.0, XA := 1);   // GTL FROM PRUB TEMPERATURE CONTROL
   TC121C : TEMP_CONTROL := (TT := -250.0, TAH_SP := 900.0, TAHH_SP := 950.0, DIFFERENCE := -302.5, TALL_TMR.PRE := 5000, TALL_TMR.ACC := 5000, TAL_TMR.PRE := 5000, TAL_TMR.ACC := 5002, TAH_TMR.PRE := 5000, TAHH_TMR.PRE := 5000, TDAH_TMR.PRE := 5000, TAHH_DEV := 945.0, TAH_DEV := 895.0, TDAH_DEV := -5.0, XA := 1);   // GTL FROM PRUC TEMPERATURE CONTROL
   TC121D : TEMP_CONTROL := (TT := -250.0, TAH_SP := 900.0, TAHH_SP := 950.0, DIFFERENCE := -302.0, TALL_TMR.PRE := 5000, TALL_TMR.ACC := 5000, TAL_TMR.PRE := 5000, TAL_TMR.ACC := 5002, TAH_TMR.PRE := 5000, TAHH_TMR.PRE := 5000, TDAH_TMR.PRE := 5000, TAHH_DEV := 945.0, TAH_DEV := 895.0, TDAH_DEV := -5.0, XA := 1);   // GTL FROM PRUD TEMPERATURE CONTROL
   TC121E : TEMP_CONTROL := (TT := -250.0, TAH_SP := 900.0, TAHH_SP := 950.0, TDAH_SP := 100.0, DIFFERENCE := -302.6, TALL_TMR.PRE := 5000, TALL_TMR.ACC := 5000, TAL_TMR.PRE := 5000, TAL_TMR.ACC := 5002, TAH_TMR.PRE := 5000, TAHH_TMR.PRE := 5000, TDAH_TMR.PRE := 5000, TAHH_DEV := 945.0, TAH_DEV := 895.0, TDAH_DEV := 95.0, XA := 1);
   TC121F : TEMP_CONTROL := (TT := -250.0, TAH_SP := 900.0, TAHH_SP := 950.0, TDAH_SP := 100.0, DIFFERENCE := -303.7, TALL_TMR.PRE := 5000, TALL_TMR.ACC := 5000, TAL_TMR.PRE := 5000, TAL_TMR.ACC := 5002, TAH_TMR.PRE := 5000, TAHH_TMR.PRE := 5000, TDAH_TMR.PRE := 5000, TAHH_DEV := 945.0, TAH_DEV := 895.0, TDAH_DEV := 95.0, XA := 1);
   TC121G : TEMP_CONTROL := (TT := -250.0, TAH_SP := 900.0, TAHH_SP := 950.0, TDAH_SP := 100.0, DIFFERENCE := -302.4, TALL_TMR.PRE := 5000, TALL_TMR.ACC := 5000, TAL_TMR.PRE := 5000, TAL_TMR.ACC := 5002, TAH_TMR.PRE := 5000, TAHH_TMR.PRE := 5000, TDAH_TMR.PRE := 5000, TAHH_DEV := 945.0, TAH_DEV := 895.0, TDAH_DEV := 95.0, XA := 1);
   TC121H : TEMP_CONTROL := (TT := -250.0, TAH_SP := 900.0, TAHH_SP := 950.0, TDAH_SP := 100.0, DIFFERENCE := -301.8, TALL_TMR.PRE := 5000, TALL_TMR.ACC := 5000, TAL_TMR.PRE := 5000, TAL_TMR.ACC := 5002, TAH_TMR.PRE := 5000, TAHH_TMR.PRE := 5000, TDAH_TMR.PRE := 5000, TAHH_DEV := 945.0, TAH_DEV := 895.0, TDAH_DEV := 95.0, XA := 1);
   TC123 : TEMP_CONTROL := (TAH_SP := 900.0, TAHH_SP := 950.0, TDAH_SP := 200.0, TAHH_DEV := 945.0, TAH_DEV := 895.0, TDAH_DEV := 195.0);
   TC123A : TEMP_CONTROL := (TT := -250.0, TAH_SP := 900.0, TAHH_SP := 950.0, TDAH_SP := 100.0, DIFFERENCE := -300.5, TAH_TMR.PRE := 5000, TAHH_TMR.PRE := 5000, TDAH_TMR.PRE := 5000, TAHH_DEV := 945.0, TAH_DEV := 895.0, TDAH_DEV := 95.0, XA := 1);   // HEAT JACKET VENT FROM PRUA TEMPERATURE CONTROL
   TC123A_SCP : SCLP := (InputMin := 4000.0, InputMax := 20000.0, ScaledMax := 1000.0, Output := -250.0);   // HEAT JACKET VENT FROM PRUA TEMPERATURE TRANSMITTER SCALER
   TC123B : TEMP_CONTROL := (TT := -250.0, TAH_SP := 900.0, TAHH_SP := 950.0, DIFFERENCE := -300.0, TAH_TMR.PRE := 5000, TAHH_TMR.PRE := 5000, TDAH_TMR.PRE := 5000, TAHH_DEV := 945.0, TAH_DEV := 895.0, TDAH_DEV := -5.0, XA := 1);
   TC123B_SCP : SCLP := (InputMin := 4000.0, InputMax := 20000.0, ScaledMax := 1000.0, Output := -250.0);   // HEAT JACKET VENT FROM PRUB TEMPERATURE TRANSMITTER SCALER
   TC123C : TEMP_CONTROL := (TT := -250.0, TAH_SP := 900.0, TAHH_SP := 950.0, DIFFERENCE := -301.5, TAH_TMR.PRE := 5000, TAHH_TMR.PRE := 5000, TDAH_TMR.PRE := 5000, TAHH_DEV := 945.0, TAH_DEV := 895.0, TDAH_DEV := -5.0, XA := 1);   // HEAT JACKET VENT FROM PRUC TEMPERATURE CONTROL
   TC123C_SCP : SCLP := (InputMin := 4000.0, InputMax := 20000.0, ScaledMax := 1000.0, Output := -250.0);   // HEAT JACKET VENT FROM PRUC TEMPERATURE TRANSMITTER SCALER
   TC123D : TEMP_CONTROL := (TT := -250.0, TAH_SP := 900.0, TAHH_SP := 950.0, TDAH_SP := 100.0, DIFFERENCE := -301.3, TAH_TMR.PRE := 5000, TAHH_TMR.PRE := 5000, TDAH_TMR.PRE := 5000, TAHH_DEV := 945.0, TAH_DEV := 895.0, TDAH_DEV := 95.0, XA := 1);   // HEAT JACKET VENT FROM PRUD TEMPERATURE TRANSMITTER
   TC123D_SCP : SCLP := (InputMin := 4000.0, InputMax := 20000.0, ScaledMax := 1000.0, Output := -250.0);   // HEAT JACKET VENT FROM PRUD TEMPERATURE TRANSMITTER SCALER
   TC123E : TEMP_CONTROL := (TT := -250.0, TAH_SP := 900.0, TAHH_SP := 950.0, TDAH_SP := 100.0, DIFFERENCE := -300.1, TAH_TMR.PRE := 5000, TAHH_TMR.PRE := 5000, TDAH_TMR.PRE := 5000, TAHH_DEV := 945.0, TAH_DEV := 895.0, TDAH_DEV := 95.0, XA := 1);
   TC123E_SCP : SCLP := (InputMin := 4000.0, InputMax := 20000.0, ScaledMax := 1000.0, Output := -250.0);
   TC123F : TEMP_CONTROL := (TT := -250.0, TAH_SP := 900.0, TAHH_SP := 950.0, TDAH_SP := 100.0, DIFFERENCE := -300.3, TAH_TMR.PRE := 5000, TAHH_TMR.PRE := 5000, TDAH_TMR.PRE := 5000, TAHH_DEV := 945.0, TAH_DEV := 895.0, TDAH_DEV := 95.0, XA := 1);
   TC123F_SCP : SCLP := (InputMin := 4000.0, InputMax := 20000.0, ScaledMax := 1000.0, Output := -250.0);
   TC123G : TEMP_CONTROL := (TT := -250.0, TAH_SP := 900.0, TAHH_SP := 950.0, TDAH_SP := 500.0, DIFFERENCE := -301.4, TAH_TMR.PRE := 5000, TAHH_TMR.PRE := 5000, TDAH_TMR.PRE := 5000, TAHH_DEV := 945.0, TAH_DEV := 895.0, TDAH_DEV := 495.0, XA := 1);
   TC123G_SCP : SCLP := (InputMin := 4000.0, InputMax := 20000.0, ScaledMax := 1000.0, Output := -250.0);
   TC123H : TEMP_CONTROL := (TT := -250.0, TAH_SP := 900.0, TAHH_SP := 950.0, TDAH_SP := 100.0, DIFFERENCE := -301.4, TAH_TMR.PRE := 5000, TAHH_TMR.PRE := 5000, TDAH_TMR.PRE := 5000, TAHH_DEV := 945.0, TAH_DEV := 895.0, TDAH_DEV := 95.0, XA := 1);
   TC123H_SCP : SCLP := (InputMin := 4000.0, InputMax := 20000.0, ScaledMax := 1000.0, Output := -250.0);
   TC135 : TEMP_CONTROL := (TT := -10.0, TALL := 1, TAL := 1, TALL_TMR.PRE := 5000, TALL_TMR.ACC := 5009, TALL_TMR.EN := 1, TALL_TMR.DN := 1, TAL_TMR.PRE := 5000, TAL_TMR.ACC := 5009, TAL_TMR.EN := 1, TAL_TMR.DN := 1, TAH_TMR.PRE := 5000, TAHH_TMR.PRE := 5000, TAHH_DEV := -5.0, TAH_DEV := -5.0, TAL_DEV := 5.0, TALL_DEV := 5.0, XA := 1, RawCounts := 3200);
   TC135_AUTO_Ons : BOOL;
   TC135_AUTO_Ons1 : BOOL;
   TC135_MANUAL_Ons : BOOL;
   TC135_PID : PID := (MAXO := 100.0);
   TC135_PID_TON : TIMER := (PRE := 500, ACC := 81);
   TC135_SCP : SCLP := (Input := 3200.0, InputMin := 4000.0, InputMax := 20000.0, ScaledMax := 200.0, Output := -10.0);
   TC136 : TEMP_CONTROL := (TT := -10.0, TALL := 1, TAL := 1, TALL_TMR.PRE := 5000, TALL_TMR.ACC := 5009, TALL_TMR.EN := 1, TALL_TMR.DN := 1, TAL_TMR.PRE := 5000, TAL_TMR.ACC := 5009, TAL_TMR.EN := 1, TAL_TMR.DN := 1, TAH_TMR.PRE := 5000, TAHH_TMR.PRE := 5000, TAHH_DEV := -5.0, TAH_DEV := -5.0, TAL_DEV := 5.0, TALL_DEV := 5.0, XA := 1, RawCounts := 3200);
   TC136_SCP : SCLP := (Input := 3200.0, InputMin := 4000.0, InputMax := 20000.0, ScaledMax := 200.0, Output := -10.0);
   TC137 : TEMP_CONTROL := (TT := -10.0, TALL := 1, TAL := 1, TALL_TMR.PRE := 5000, TALL_TMR.ACC := 5009, TALL_TMR.EN := 1, TALL_TMR.DN := 1, TAL_TMR.PRE := 5000, TAL_TMR.ACC := 5009, TAL_TMR.EN := 1, TAL_TMR.DN := 1, TAH_TMR.PRE := 5000, TAHH_TMR.PRE := 5000, TAHH_DEV := -5.0, TAH_DEV := -5.0, TAL_DEV := 5.0, TALL_DEV := 5.0, XA := 1, RawCounts := 3200);
   TC137_SCP : SCLP := (Input := 3200.0, InputMin := 4000.0, InputMax := 20000.0, ScaledMax := 200.0, Output := -10.0);
   TC215 : TEMP_CONTROL := (AUTO := 1, MAN_SP := 100.0, AUTO_SP := 60.0, CO := 100.0, FB := 100.0, TT := 67.537506, TALL_SP := 35.0, TAL_SP := 40.0, TAH_SP := 120.0, TAHH_SP := 130.0, TALL_TMR.PRE := 5000, TAL_TMR.PRE := 5000, TAH_TMR.PRE := 5000, TAHH_TMR.PRE := 5000, TAHH_DEV := 125.0, TAH_DEV := 115.0, TAL_DEV := 45.0, TALL_DEV := 40.0, RawCounts := 7602);   // OVERHEAD CONDENSER CHILLED WATER TEMPERATURE TRANSMITTER CONTROL
   TC215_AUTO_ONS1 : BOOL := 1;
   TC215_MANUAL_ONS1 : BOOL;
   TC215_SCP : SCLP := (Input := 7602.0, InputMin := 4000.0, InputMax := 20000.0, ScaledMax := 300.0, Output := 67.537506);   // OVERHEAD CONDENSER CHILLED WATER TEMPERATURE TRANSMITTER SCALER
   TC216 : TEMP_CONTROL := (TT := 65.34375, RawCounts := 7485);   // OVERHEAD CONDENSER BASIN TEMPERATURE CONTROL
   TC217 : TEMP_CONTROL := (TT := 66.58125, RawCounts := 7551);   // OVERHEAD CONDENSED CHILLED WATER RETURN TEMPERATURE CONTROL
   TC218 : TEMP_CONTROL := (TT := 66.52501, RawCounts := 7548);   // OVERHEAD CONDENSER CHILLED WATER SUPPLY TEMPERATURE CONTROL
   TC306 : TEMP_CONTROL;
   TC313A : TEMP_CONTROL := (AUTO := 1, MAN_SP := 50.0, AUTO_SP := 135.0, PID_CO := 50.0, TT := 64.01251, TALL_SP := 115.0, TAL_SP := 120.0, TAH_SP := 155.0, TAHH_SP := 165.0, TALL := 1, TAL := 1, TALL_TMR.PRE := 5000, TALL_TMR.ACC := 5008, TALL_TMR.EN := 1, TALL_TMR.DN := 1, TAL_TMR.PRE := 5000, TAL_TMR.ACC := 5008, TAL_TMR.EN := 1, TAL_TMR.DN := 1, TAH_TMR.PRE := 5000, TAHH_TMR.PRE := 5000, TAHH_DEV := 160.0, TAH_DEV := 150.0, TAL_DEV := 125.0, TALL_DEV := 120.0, RawCounts := 7414);   // PRIMARY COALESCER SEPARATOR TEMPERATURE CONTROL
   TC313A_AUTO_Ons : BOOL := 1;
   TC313A_AUTO_Ons1 : BOOL;
   TC313A_HeaterDisabled : BOOL := 1;
   TC313A_MANUAL_Ons : BOOL;
   TC313A_NoPumpsRunningAlm : BOOL;
   TC313A_START_TON : TIMER := (PRE := 5000);
   TC313B : TEMP_CONTROL := (TT := -14.999996, TALL_SP := 110.0, TAL_SP := 115.0, TAH_SP := 280.0, TAHH_SP := 300.0, TALL := 1, TAL := 1, TALL_TMR.PRE := 5000, TALL_TMR.ACC := 5001, TALL_TMR.EN := 1, TALL_TMR.DN := 1, TAL_TMR.PRE := 5000, TAL_TMR.ACC := 5001, TAL_TMR.EN := 1, TAL_TMR.DN := 1, TAH_TMR.PRE := 5000, TAHH_TMR.PRE := 5000, TAHH_DEV := 295.0, TAH_DEV := 275.0, TAL_DEV := 120.0, TALL_DEV := 115.0, XA := 1, RawCounts := 3200);   // PRIMARY COALESCER SHELL TEMPERATURE CONTROL
   TC319 : TEMP_CONTROL := (AUTO := 1, AUTO_SP := 100.0, TT := -14.999996, TALL_SP := 90.0, TAL_SP := 100.0, TAH_SP := 280.0, TAHH_SP := 300.0, TALL := 1, TAL := 1, TALL_TMR.PRE := 5000, TALL_TMR.ACC := 5009, TALL_TMR.EN := 1, TALL_TMR.DN := 1, TAL_TMR.PRE := 5000, TAL_TMR.ACC := 5009, TAL_TMR.EN := 1, TAL_TMR.DN := 1, TAH_TMR.PRE := 5000, TAHH_TMR.PRE := 5000, TAHH_DEV := 295.0, TAH_DEV := 275.0, TAL_DEV := 105.0, TALL_DEV := 95.0, XA := 1, RawCounts := 3200);   // COALESCER OIL CHAMBER PROCESS TEMPERATURE CONTROL
   TC319_AUTO_Ons : BOOL := 1;
   TC319_AUTO_Ons1 : BOOL;
   TC319_Disabled : BOOL;
   TC319_FlowComplete : BOOL;
   TC319_HeaterDisabled : BOOL := 1;
   TC319_MANUAL_Ons : BOOL;
   TC319_NoPumpsRunningAlm : BOOL;
   TC319_START_TON : TIMER := (PRE := 5000);
   TC319A : TEMP_CONTROL := (TT := -14.999996, TALL := 1, TAL := 1, TALL_TMR.PRE := 5000, TALL_TMR.ACC := 5009, TALL_TMR.EN := 1, TALL_TMR.DN := 1, TAL_TMR.PRE := 5000, TAL_TMR.ACC := 5009, TAL_TMR.EN := 1, TAL_TMR.DN := 1, TAH_TMR.PRE := 5000, TAHH_TMR.PRE := 5000, TAHH_DEV := -5.0, TAH_DEV := -5.0, TAL_DEV := 5.0, TALL_DEV := 5.0, XA := 1, RawCounts := 3200);   // COALESCER OIL CHAMBER SHEATH TEMPERATURE
   TC320 : TEMP_CONTROL := (TT := 65.60626, TAH := 1, TAHH := 1, TALL_TMR.PRE := 5000, TAL_TMR.PRE := 5000, TAH_TMR.PRE := 5000, TAH_TMR.ACC := 5008, TAH_TMR.EN := 1, TAH_TMR.DN := 1, TAHH_TMR.PRE := 5000, TAHH_TMR.ACC := 5008, TAHH_TMR.EN := 1, TAHH_TMR.DN := 1, TAHH_DEV := -5.0, TAH_DEV := -5.0, TAL_DEV := 5.0, TALL_DEV := 5.0, RawCounts := 7499);   // COALESCER OIL CHAMBER SHELL TEMPERATURE TRANSMITTER CONTROL
   TC321A : TEMP_CONTROL := (TT := 64.10626, TAH_SP := 160.0, TAHH_SP := 180.0, TALL_TMR.PRE := 5000, TAL_TMR.PRE := 5000, TAH_TMR.PRE := 5000, TAHH_TMR.PRE := 5000, TAHH_DEV := 175.0, TAH_DEV := 155.0, TAL_DEV := 5.0, TALL_DEV := 5.0, RawCounts := 7419);   // COALESCER OIL CHAMBER TRANSFER PUMP A TEMPERATURE TRANSMITTER
   TC321B : TEMP_CONTROL := (TT := 64.8, TAH_SP := 160.0, TAHH_SP := 180.0, TALL_TMR.PRE := 5000, TAL_TMR.PRE := 5000, TAH_TMR.PRE := 5000, TAHH_TMR.PRE := 5000, TAHH_DEV := 175.0, TAH_DEV := 155.0, TAL_DEV := 5.0, TALL_DEV := 5.0, RawCounts := 7456);   // COALESCER OIL CHAMBER TRANSFER PUMP B TEMPERATURE TRANSMITTER
   TC406 : TEMP_CONTROL := (AUTO := 1, MAN_SP := 20.0, AUTO_SP := 140.0, TT := 66.375, TALL_SP := 90.0, TAL_SP := 130.0, TAH_SP := 150.0, TAHH_SP := 150.0, TALL := 1, TAL := 1, TALL_TMR.PRE := 5000, TALL_TMR.ACC := 5009, TALL_TMR.EN := 1, TALL_TMR.DN := 1, TAL_TMR.PRE := 5000, TAL_TMR.ACC := 5009, TAL_TMR.EN := 1, TAL_TMR.DN := 1, TAH_TMR.PRE := 5000, TAHH_TMR.PRE := 5000, TAHH_DEV := 155.0, TAH_DEV := 155.0, TAL_DEV := 125.0, TALL_DEV := 85.0, RawCounts := 7540);   // PROCESS WATER POST HX TEMPERATURE CONTROL
   TC406_AUTO_ONS1 : BOOL := 1;
   TC406_LockOut : BOOL := 1;
   TC406_MANUAL_ONS1 : BOOL;
   TC406_SCP : SCLP := (Input := 7540.0, InputMin := 4000.0, InputMax := 20000.0, ScaledMax := 300.0, Output := 66.375);   // PROCESS WATER POST HX TEMPERATURE TRANSMITTER SCALER
   TC409 : TEMP_CONTROL := (TT := 66.99376, TAH := 1, TAHH := 1, TALL_TMR.PRE := 5000, TAL_TMR.PRE := 5000, TAH_TMR.PRE := 5000, TAH_TMR.ACC := 5009, TAH_TMR.EN := 1, TAH_TMR.DN := 1, TAHH_TMR.PRE := 5000, TAHH_TMR.ACC := 5009, TAHH_TMR.EN := 1, TAHH_TMR.DN := 1, TAHH_DEV := -5.0, TAH_DEV := -5.0, TAL_DEV := 5.0, TALL_DEV := 5.0, RawCounts := 7573);   // HX COOLING WATER SUPPLY TEMPERATURE CONTROL
   TC409_SCP : SCLP := (Input := 7571.0, InputMin := 4000.0, InputMax := 20000.0, ScaledMax := 300.0, Output := 66.95625);   // HX COOLING WATER SUPPLY TEMPERATURE TRANSMITTER SCALER
   TC410 : TEMP_CONTROL := (TT := 66.46875, TAH := 1, TAHH := 1, TALL_TMR.PRE := 5000, TAL_TMR.PRE := 5000, TAH_TMR.PRE := 5000, TAH_TMR.ACC := 5009, TAH_TMR.EN := 1, TAH_TMR.DN := 1, TAHH_TMR.PRE := 5000, TAHH_TMR.ACC := 5009, TAHH_TMR.EN := 1, TAHH_TMR.DN := 1, TAHH_DEV := -5.0, TAH_DEV := -5.0, TAL_DEV := 5.0, TALL_DEV := 5.0, RawCounts := 7545);   // HX COOLING WATER RETURN TEMPERATURE CONTROL
   TC410_SCP : SCLP := (Input := 7545.0, InputMin := 4000.0, InputMax := 20000.0, ScaledMax := 300.0, Output := 66.46875);   // HX COOLING WATER RETURN TEMPERATURE TRANSMITTER SCALER
   TCP_GetAll : TCPGetAllConfig := (IPAddress := 16#c0a8_1446, SubNetMask := 16#ffff_0000);
   TCP_SetAll : TCPSetAllConfig := (IPAddress := 16#c0a8_3246, SubNetMask := 16#ffff_ff00, Gateway := 16#c0a8_3201);
   TCV108_SCP : SCLP := (Input := 3200.0, InputMin := 4000.0, InputMax := 20000.0, ScaledMax := 100.0, Output := -5.0);
   TCV215_PID : PID := (CTL := 33591936, CA := 1, INI := 1, OLH := 1, DVPA := 1, PVHA := 1, SP := 60.0, KP := 20.0, KI := 2.0, MAXS := 4000.0, SO := 100.0, MAXO := 100.0, MINO := 30.0, UPD := 0.1, PV := 67.537506, ERR := 7.537506, OUT := 100.0, MAXI := 4000.0, MAXCV := 100.0, MAXTIE := 4095.0, DATA[0] := 97.391594, DATA[1] := 27.015003, DATA[2] := 67.537506, DATA[3] := 7.537506, DATA[4] := 60.0, DATA[5] := 0.025, DATA[6] := 1.0, DATA[7] := 1.6, DATA[8] := 20.0, DATA[9] := 2.0, DATA[11] := 20.0, DATA[12] := 2.0, DATA[15] := 1.0, DATA[16] := 0.024420025);
   TCV215_SCP : SCLP := (Input := 100.0, InputMax := 100.0, ScaledMin := 4000.0, ScaledMax := 20000.0, Output := 20000.0);   // CONDENSER CHILLED WATER VALVE CONTROL OUTPUT
   TCV406 : TEMP_CONTROL := (MANUAL := 1, MAN_SP := 20.0, TT := 44.2125);
   TCV406_SCP : SCLP := (InputMax := 100.0, ScaledMin := 4000.0, ScaledMax := 20000.0, Output := 4000.0);   // QUENCH CONDITIONING HX COOLING WATER CONTROL VALVE
   TCV406_SP : SCLP := (Input := 3200.0, InputMin := 4000.0, InputMax := 20000.0, ScaledMax := 100.0, Output := -5.0);
   TEMP_DINT : DINT := 4000;
   Test : INT[500] := ([10] := -25029, [11] := 21064, [12] := 13908, [13] := 11826, [14] := 13360, [15] := 14128, [16] := 13360, [17] := 14128, [18] := 12592, [19] := -32512, [20] := -32542, [21] := -32542, [24] := 784, [25] := 3, [26] := 4, [28] := 4, [29] := 4, [31] := 18142, [32] := 12938, [34] := 64, [35] := 64, [37] := 1, [38] := 62, [39] := 62, [42] := 23481, [45] := -1, [90] := 62, [100] := -10864, [101] := 16546, [102] := -18748, [103] := 16601, [104] := -18748, [105] := 16601, [108] := 11441, [109] := 17222, [110] := 16384, [111] := 14649, [112] := 9273);
   testMSG : MESSAGE;
        MessageParameters(ServiceCode := 16#004c, LocalElement := MyDint, ...)
   TestyBit : DINT := 6684867;
   TIMER : TIMER[50] := ([0].PRE := 5000, [1].PRE := 60000, [1].ACC := 827, [2].PRE := 60000, [2].ACC := 827, [2].EN := 1, [2].TT := 1, [3].PRE := 2000, [5].PRE := 60000, [5].ACC := 827, [5].EN := 1, [5].TT := 1, [6].PRE := 2000, [7].PRE := 60000, [7].ACC := 1842, [7].EN := 1, [7].TT := 1, [8].PRE := 2000, [9].PRE := 60000, [9].ACC := 827, [9].EN := 1, [9].TT := 1, [10].PRE := 2000, [11].PRE := 5000, [12].PRE := 5000, [12].EN := 1, [12].TT := 1, [13].PRE := 5000, [15].PRE := 5000, [15].ACC := 5009, [15].EN := 1, [15].DN := 1, [16].PRE := 5000, [17].PRE := 5000, [17].ACC := 5009, [17].EN := 1, [17].DN := 1);   // HX A TIMER FOR START
        [0]   // P101B TIMER
        [1]   // P303B TIMER
        [5]   // PRUB HB TIMER ON
        [6]   // PRUC HB TIMER OFF
        [2]   // PRUA HB TIMER ON
        [3]   // PRUA TIMER OFF
        [7]   // PRUC HB TIMER ON
        [8]   // PRUC HB TIMER OFF
        [9]   // PRUD HB TIMER ON
        [10]   // PRUD HB TIMER OFF
   TMR_CRIT_FAULT : DINT := 300000;
   TMR_FAULT : DINT := 5000;
   tog : BOOL := 1;
   TT101A_SCP : SCLP := (Input := 7390.0, InputMin := 4000.0, InputMax := 20000.0, ScaledMax := 300.0, Output := 63.5625);   // QUENCH BASIN TRANSFER BASIN A TEMPERATURE TRANSMITTER SCALER
   TT101B_SCP : SCLP := (Input := 7410.0, InputMin := 4000.0, InputMax := 20000.0, ScaledMax := 300.0, Output := 63.9375);   // QUENCH BASIN TRANSFER BASIN B TEMPERATURE TRANSMITTER SCALER
   TT108_SCP : SCLP := (Input := 7712.0, InputMin := 4000.0, InputMax := 20000.0, ScaledMax := 300.0, Output := 69.600006);   // QUENCH TOWER EXIT GAS TEMPERATURE TRANSMITTER SCALER
   TT114A_SCP : SCLP := (Input := 7426.0, InputMin := 4000.0, InputMax := 20000.0, ScaledMax := 300.0, Output := 64.2375);   // QUENCH BASIN SHELL TEMPERATURE TRANSMITTER SCALER
   TT114B_SCP : SCLP := (Input := 7425.0, InputMin := 4000.0, InputMax := 20000.0, ScaledMax := 300.0, Output := 64.21875);   // QUENCH BASIN LIQUID TEMPERATURE TRANSMITTER SCALER
   TT121A_SCP : SCLP := (InputMin := 4000.0, InputMax := 20000.0, ScaledMax := 1000.0, Output := -250.0);   // GTL FROM PRUA TEMPERATURE TRANSMITTER SCALER
   TT121B_SCP : SCLP := (InputMin := 4000.0, InputMax := 20000.0, ScaledMax := 1000.0, Output := -250.0);
   TT121C_SCP : SCLP := (InputMin := 4000.0, InputMax := 20000.0, ScaledMax := 1000.0, Output := -250.0);
   TT121D_SCP : SCLP := (InputMin := 4000.0, InputMax := 20000.0, ScaledMax := 1000.0, Output := -250.0);
   TT121E_SCP : SCLP := (InputMin := 4000.0, InputMax := 20000.0, ScaledMax := 1000.0, Output := -250.0);
   TT121F_SCP : SCLP := (InputMin := 4000.0, InputMax := 20000.0, ScaledMax := 1000.0, Output := -250.0);   // GTL FROM PRUB TEMPERATURE TRANSMITTER SCALER
   TT121G_SCP : SCLP := (InputMin := 4000.0, InputMax := 20000.0, ScaledMax := 1000.0, Output := -250.0);   // GTL FROM PRUC TEMPERATURE TRANSMITTER SCALER
   TT121H_SCP : SCLP := (InputMin := 4000.0, InputMax := 20000.0, ScaledMax := 1000.0, Output := -250.0);   // GTL FROM PRUD TEMPERATURE TRANSMITTER SCALER
   TT215_SCP : SCLP := (Input := 6508.0, InputMin := 4000.0, InputMax := 20000.0, ScaledMax := 300.0, Output := 47.025);
   TT216_SCP : SCLP := (Input := 7482.0, InputMin := 4000.0, InputMax := 20000.0, ScaledMax := 300.0, Output := 65.287506);   // OVERHEAD CONDENSER BASIN TEMPERATURE TRANSMITTER SCALER
   TT217_SCP : SCLP := (Input := 7551.0, InputMin := 4000.0, InputMax := 20000.0, ScaledMax := 300.0, Output := 66.58125);   // OVERHEAD CONDENSED CHILLED WATER RETURN TEMPERATURE TRANSMITTER
   TT218_SCP : SCLP := (Input := 7548.0, InputMin := 4000.0, InputMax := 20000.0, ScaledMax := 300.0, Output := 66.52501);   // OVERHEAD CONDENSER CHILLED WATER SUPPLY TEMPERATURE SCALER
   TT313A_SCP : SCLP := (Input := 7414.0, InputMin := 4000.0, InputMax := 20000.0, ScaledMax := 300.0, Output := 64.01251);   // PRIMARY COALESCER SEPARATOR TEMPERATURE TRANSMITTER SCALER
   TT313B_SCP : SCLP := (Input := 3200.0, InputMin := 4000.0, InputMax := 20000.0, ScaledMax := 300.0, Output := -14.999996);   // PRIMARY COALESCER SHELL TEMPERATURE TRANSMITTER SCALER
   TT319_SCP : SCLP := (Input := 3200.0, InputMin := 4000.0, InputMax := 20000.0, ScaledMax := 300.0, Output := -14.999996);   // COALESCER OIL CHAMBER SHELL TEMPERATURE TRANSMITTER SCALER
   TT319A_SCP : SCLP := (Input := 3200.0, InputMin := 4000.0, InputMax := 20000.0, ScaledMax := 300.0, Output := -14.999996);
   TT320_SCP : SCLP := (Input := 7498.0, InputMin := 4000.0, InputMax := 20000.0, ScaledMax := 300.0, Output := 65.58751);   // COALESCER OIL CHAMBER SHELL TEMPERATURE TRANSMITTER SCALER
   TT321A_SCP : SCLP := (Input := 7419.0, InputMin := 4000.0, InputMax := 20000.0, ScaledMax := 300.0, Output := 64.10626);   // COALESCER OIL CHAMBER TRANSFER PUMP A TEMPERATURE TRANSMITTER SCALER
   TT321B_SCP : SCLP := (Input := 7457.0, InputMin := 4000.0, InputMax := 20000.0, ScaledMax := 300.0, Output := 64.818756);   // COALESCER OIL CHAMBER TRANSFER PUMP B TEMPERATURE TRANSMITTER
   UTIL_1 : INT;   // ONE SHOTS FOR UTILITIES
   UTIL_CON : INT[2];   // UTILITIES CONNECTION WORD 0 = ALARM MASTER WORD 1 = POWER STATUS
        [0].2   // UTILITIES CSS_START_DISABLE
        [1]   // UTILITIES POWER STATUS
        [1].0   // HOUSE POWER OK
        [1].1   // GENERATOR STATUS
        [0]   // UTILITIES AlarmMaster
        [0].4   // UTILITIES PRU_RUN_DISABLE (ECool)
        [0].3   // UTILITIES PRU_START_DISABLE
        [0].0   // UTILITIES MESSAGE ALARM
        [0].1   // UTILITIES WARNING ALARM
   UTIL_READ : INT[30];   // UTILITIES SYSTEM
   UTIL_READ_MSG : MESSAGE;
        MessageParameters(ServiceCode := 16#004c, LocalElement := UTIL_CON[0], ...)
   UTL_AlarmMaster : DINT := 3;
   UTL_Comms : DINT[3] := ([0] := 3, [1] := 35, [2] := 60);
        [0]   // UTILITIES AlarmMaster
        [1].1   // HOUSE POWER OK
        [1]   // UTILITIES POWER STATUS
        [0].0   // UTILITIES MESSAGE ALARM
        [0].1   // UTILITIES WARNING ALARM
        [0].2   // UTILITIES CSS_START_DISABLE ALARM
        [0].3   // UTILITIES PRU_START_DISABLE ALARM
        [0].4   // UTILITIES PRU_RUN_DISABLE ALARM
        [1].2   // GENERATOR STATUS
        [1].0   // UTILITY PLC HEARTBEAT STATUS
        [2]   // COMMS LOSS ALARM SP (Sec)
        [1].3   // WRS Cannot Accept Water (0=OK, 1=Alarm)
        [1].4   // FIRE SYSTEM FLOW ALARM
        [1].5   // OPTION F1 OCCUPANCY 0=DISABLED 1=ENABLED
   UTL_CommsLossAlm : BOOL := 1;
   UTL_HeartbeatTimer : TIMER := (PRE := 60000, ACC := 60000, EN := 1, DN := 1);
   UTL_READ_MSG : MESSAGE;
        MessageParameters(ServiceCode := 16#004c, LocalElement := UTL_Comms[0], ...)
   WarmBoot : BOOL;
   Warnings : DINT;
   WRS_OK : BOOL := 1;
END_VAR

PROGRAM MainProgram   (* main routine MainRoutine *)
VAR
   AT102A_SCP : SCLP := (Input := 3200.0, InputMin := 4000.0, InputMax := 20000.0, ScaledMax := 1000.0, Output := -50.0);   // QUENCH WATER CONDUCTIVITY TRANSMITTER SCALER (0-100 milli Siemens)
   CSS_OK_TO_RUN_latch : BOOL := 1;
   CSS_OK_TO_RUN_os_tb : BOOL := 1;
   CSS_SHUT_PALL : BOOL;
   DLM1 : BOOL;
   FCV141 : ValveControl_TwoWay;
   HX433B_OPEN : BOOL;
   MV433A_OPEN : BOOL;
   MV433B_OPEN : BOOL;
   P302A_QI_AUTO_OS : BOOL := 1;
   P302A_QI_MAN_OS : BOOL;
   P302B_QI_AUTO_ONS1 : BOOL := 1;
   PRUA_READ_MSG_ER_CTU : COUNTER;
   PRUC_HeartbeatCommsLoss_latch : BOOL := 1;
   PRUC_HeartbeatCommsLoss_os_tb : BOOL;
   PRUE_READ_MSG_ER_CTU : COUNTER;
   PRUF_READ_MSG_ER_CTU : COUNTER;
   PRUG_READ_MSG_ER_CTU : COUNTER;
   PRUH_READ_MSG_ER_CTU : COUNTER;
   TESTOUT : REAL := 10.0;
   Toggle : BOOL := 1;
   UTL_Comms_ons : BOOL;
   UTL_CommsLossAlm_latch : BOOL := 1;
   UTL_CommsLossAlm_os_tb : BOOL;
END_VAR

ROUTINE A0_Serialize_Me   (* ladder *)
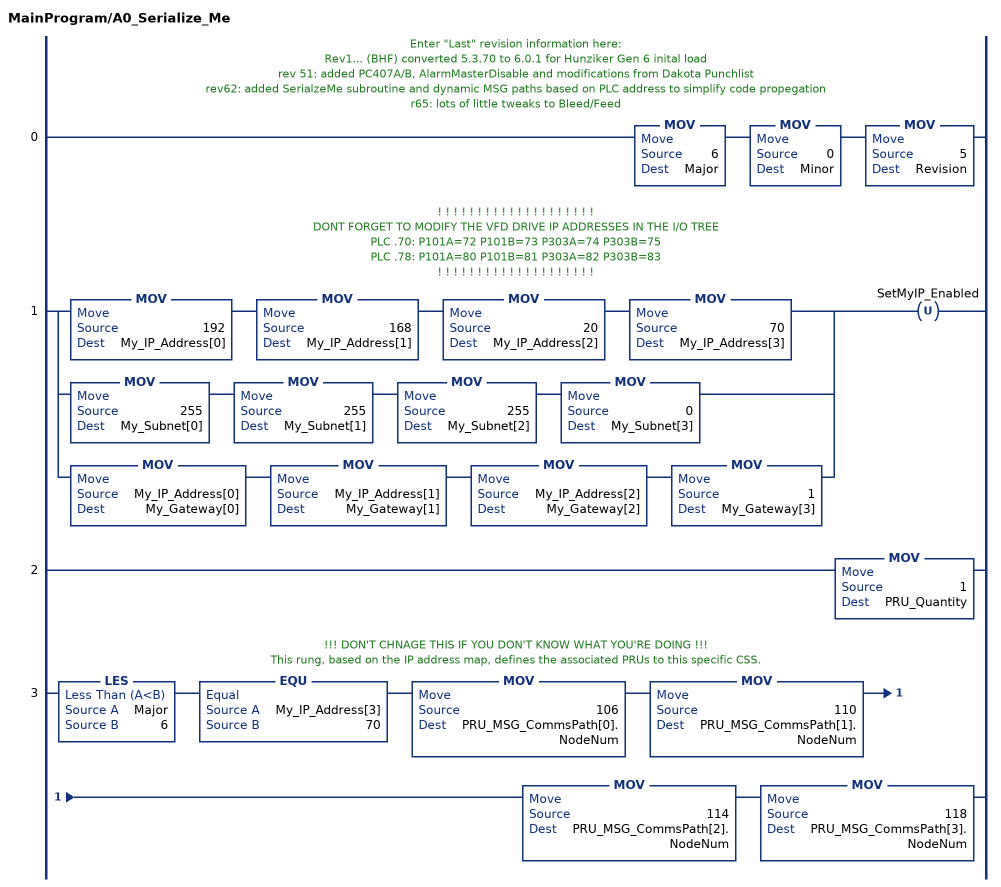
   // Enter "Last" revision information here:
   // Rev1... (BHF) converted 5.3.70 to 6.0.1 for Hunziker Gen 6 inital load
   // rev 51: added PC407A/B, AlarmMasterDisable and modifications from Dakota Punchlist
   // rev62: added SerialzeMe subroutine and dynamic MSG paths based on PLC address to simplify code propegation
   // r65: lots of little tweaks to Bleed/Feed
   0: MOV(6,Major)MOV(0,Minor)MOV(5,Revision);
   // ! ! ! ! ! ! ! ! ! ! ! ! ! ! ! ! ! ! ! !
   // DONT FORGET TO MODIFY THE VFD DRIVE IP ADDRESSES IN THE I/O TREE
   // PLC .70: P101A=72 P101B=73 P303A=74 P303B=75
   // PLC .78: P101A=80 P101B=81 P303A=82 P303B=83
   // ! ! ! ! ! ! ! ! ! ! ! ! ! ! ! ! ! ! ! !
   1: [MOV(192,My_IP_Address[0]) MOV(168,My_IP_Address[1]) MOV(20,My_IP_Address[2]) MOV(70,My_IP_Address[3]) ,MOV(255,My_Subnet[0]) MOV(255,My_Subnet[1]) MOV(255,My_Subnet[2]) MOV(0,My_Subnet[3]) ,MOV(My_IP_Address[0],My_Gateway[0]) MOV(My_IP_Address[1],My_Gateway[1]) MOV(My_IP_Address[2],My_Gateway[2]) MOV(1,My_Gateway[3]) ]OTU(SetMyIP_Enabled);
   2: MOV(1,PRU_Quantity);
   // !!! DON'T CHNAGE THIS IF YOU DON'T KNOW WHAT YOU'RE DOING !!!
   // This rung, based on the IP address map, defines the associated PRUs to this specific CSS.
   3: LES(Major,6)EQU(My_IP_Address[3],70)MOV(106,PRU_MSG_CommsPath[0].NodeNum)MOV(110,PRU_MSG_CommsPath[1].NodeNum)MOV(114,PRU_MSG_CommsPath[2].NodeNum)MOV(118,PRU_MSG_CommsPath[3].NodeNum);
END_ROUTINE

ROUTINE A1a_MAI   (* ladder *)
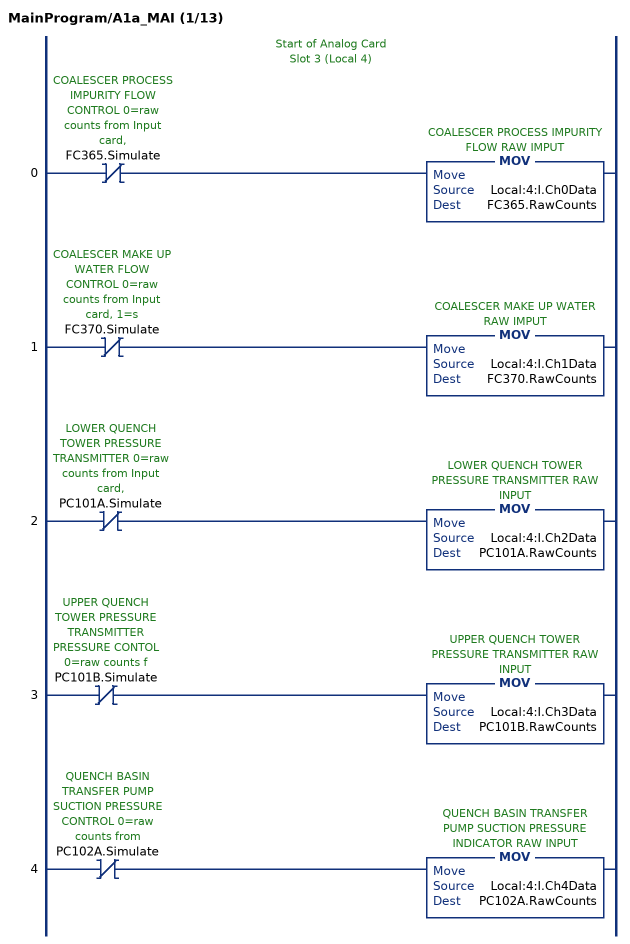
   // Start of Analog Card
   // Slot 3 (Local 4)
   0: XIO(FC365.Simulate)MOV(Local:4:I.Ch0Data,FC365.RawCounts);
   1: XIO(FC370.Simulate)MOV(Local:4:I.Ch1Data,FC370.RawCounts);
   2: XIO(PC101A.Simulate)MOV(Local:4:I.Ch2Data,PC101A.RawCounts);
   3: XIO(PC101B.Simulate)MOV(Local:4:I.Ch3Data,PC101B.RawCounts);
   4: XIO(PC102A.Simulate)MOV(Local:4:I.Ch4Data,PC102A.RawCounts);
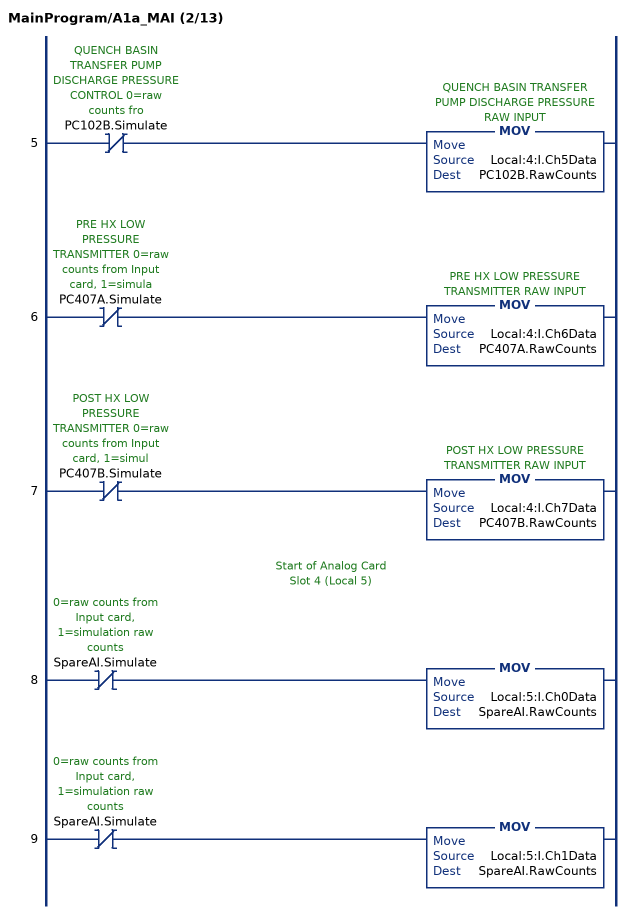
   5: XIO(PC102B.Simulate)MOV(Local:4:I.Ch5Data,PC102B.RawCounts);
   6: XIO(PC407A.Simulate)MOV(Local:4:I.Ch6Data,PC407A.RawCounts);
   7: XIO(PC407B.Simulate)MOV(Local:4:I.Ch7Data,PC407B.RawCounts);
   // Start of Analog Card
   // Slot 4 (Local 5)
   8: XIO(SpareAI.Simulate)MOV(Local:5:I.Ch0Data,SpareAI.RawCounts);
   9: XIO(SpareAI.Simulate)MOV(Local:5:I.Ch1Data,SpareAI.RawCounts);
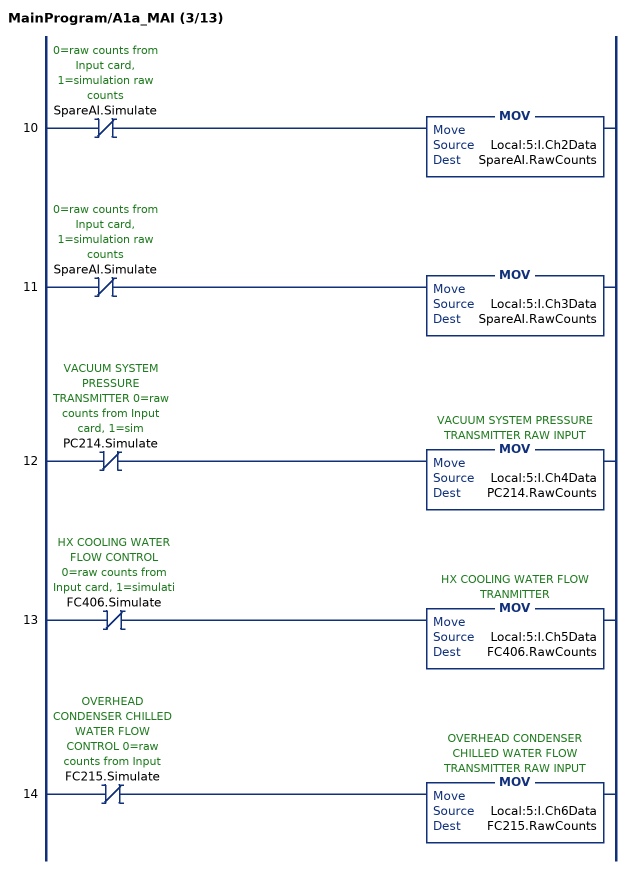
   10: XIO(SpareAI.Simulate)MOV(Local:5:I.Ch2Data,SpareAI.RawCounts);
   11: XIO(SpareAI.Simulate)MOV(Local:5:I.Ch3Data,SpareAI.RawCounts);
   12: XIO(PC214.Simulate)MOV(Local:5:I.Ch4Data,PC214.RawCounts);
   13: XIO(FC406.Simulate)MOV(Local:5:I.Ch5Data,FC406.RawCounts);
   14: XIO(FC215.Simulate)MOV(Local:5:I.Ch6Data,FC215.RawCounts);
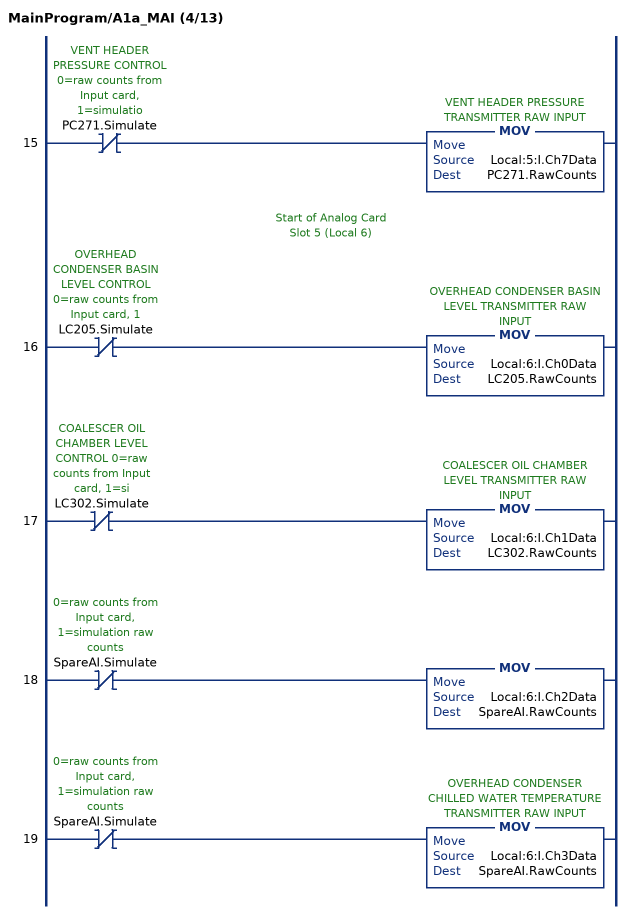
   15: XIO(PC271.Simulate)MOV(Local:5:I.Ch7Data,PC271.RawCounts);
   // Start of Analog Card
   // Slot 5 (Local 6)
   16: XIO(LC205.Simulate)MOV(Local:6:I.Ch0Data,LC205.RawCounts);
   17: XIO(LC302.Simulate)MOV(Local:6:I.Ch1Data,LC302.RawCounts);
   18: XIO(SpareAI.Simulate)MOV(Local:6:I.Ch2Data,SpareAI.RawCounts);
   19: XIO(SpareAI.Simulate)MOV(Local:6:I.Ch3Data,SpareAI.RawCounts);
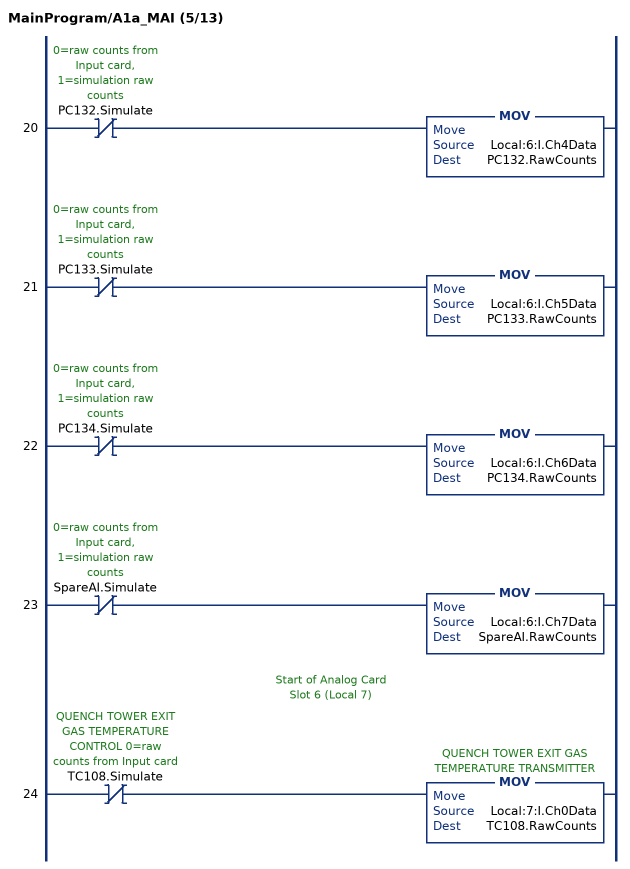
   20: XIO(PC132.Simulate)MOV(Local:6:I.Ch4Data,PC132.RawCounts);
   21: XIO(PC133.Simulate)MOV(Local:6:I.Ch5Data,PC133.RawCounts);
   22: XIO(PC134.Simulate)MOV(Local:6:I.Ch6Data,PC134.RawCounts);
   23: XIO(SpareAI.Simulate)MOV(Local:6:I.Ch7Data,SpareAI.RawCounts);
   // Start of Analog Card
   // Slot 6 (Local 7)
   24: XIO(TC108.Simulate)MOV(Local:7:I.Ch0Data,TC108.RawCounts);
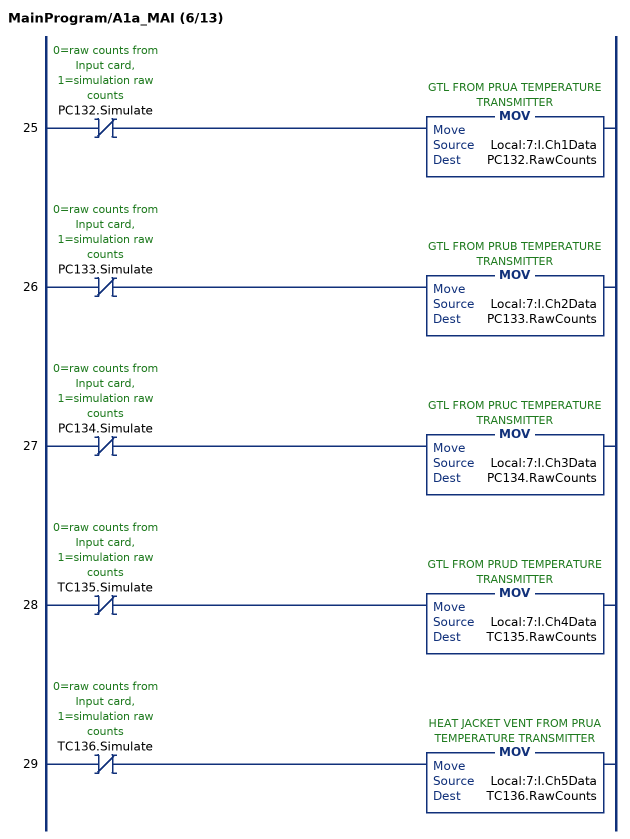
   25: XIO(PC132.Simulate)MOV(Local:7:I.Ch1Data,PC132.RawCounts);
   26: XIO(PC133.Simulate)MOV(Local:7:I.Ch2Data,PC133.RawCounts);
   27: XIO(PC134.Simulate)MOV(Local:7:I.Ch3Data,PC134.RawCounts);
   28: XIO(TC135.Simulate)MOV(Local:7:I.Ch4Data,TC135.RawCounts);
   29: XIO(TC136.Simulate)MOV(Local:7:I.Ch5Data,TC136.RawCounts);
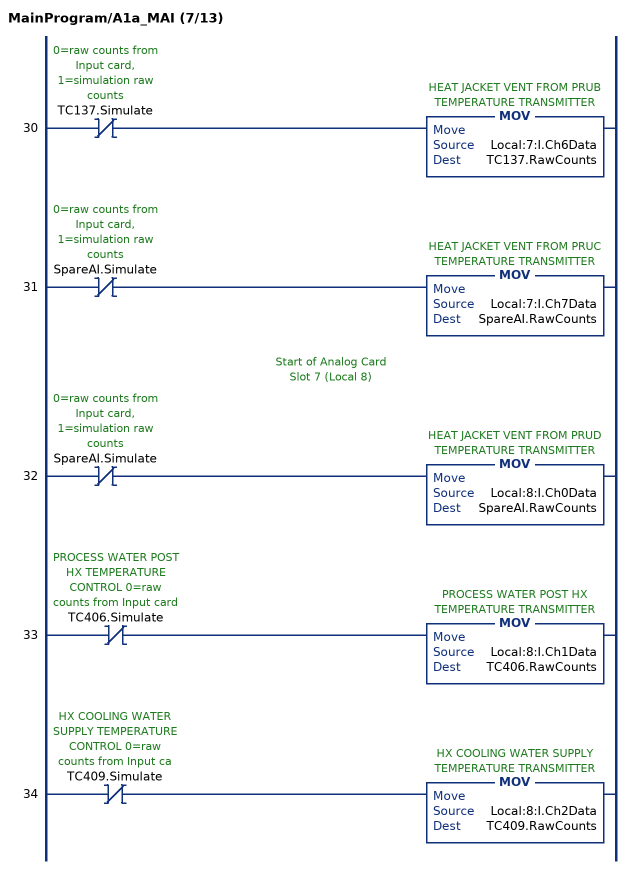
   30: XIO(TC137.Simulate)MOV(Local:7:I.Ch6Data,TC137.RawCounts);
   31: XIO(SpareAI.Simulate)MOV(Local:7:I.Ch7Data,SpareAI.RawCounts);
   // Start of Analog Card
   // Slot 7 (Local 8)
   32: XIO(SpareAI.Simulate)MOV(Local:8:I.Ch0Data,SpareAI.RawCounts);
   33: XIO(TC406.Simulate)MOV(Local:8:I.Ch1Data,TC406.RawCounts);
   34: XIO(TC409.Simulate)MOV(Local:8:I.Ch2Data,TC409.RawCounts);
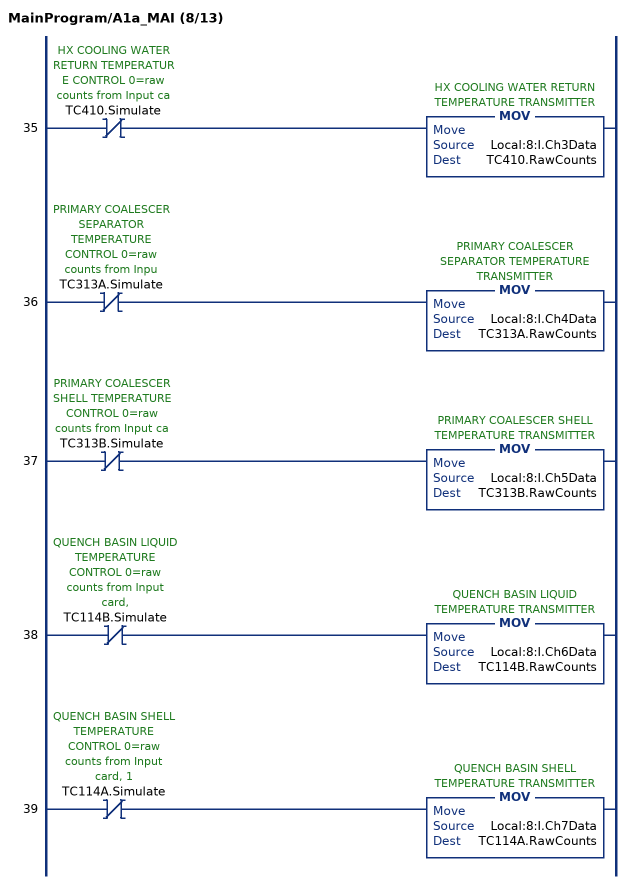
   35: XIO(TC410.Simulate)MOV(Local:8:I.Ch3Data,TC410.RawCounts);
   36: XIO(TC313A.Simulate)MOV(Local:8:I.Ch4Data,TC313A.RawCounts);
   37: XIO(TC313B.Simulate)MOV(Local:8:I.Ch5Data,TC313B.RawCounts);
   38: XIO(TC114B.Simulate)MOV(Local:8:I.Ch6Data,TC114B.RawCounts);
   39: XIO(TC114A.Simulate)MOV(Local:8:I.Ch7Data,TC114A.RawCounts);
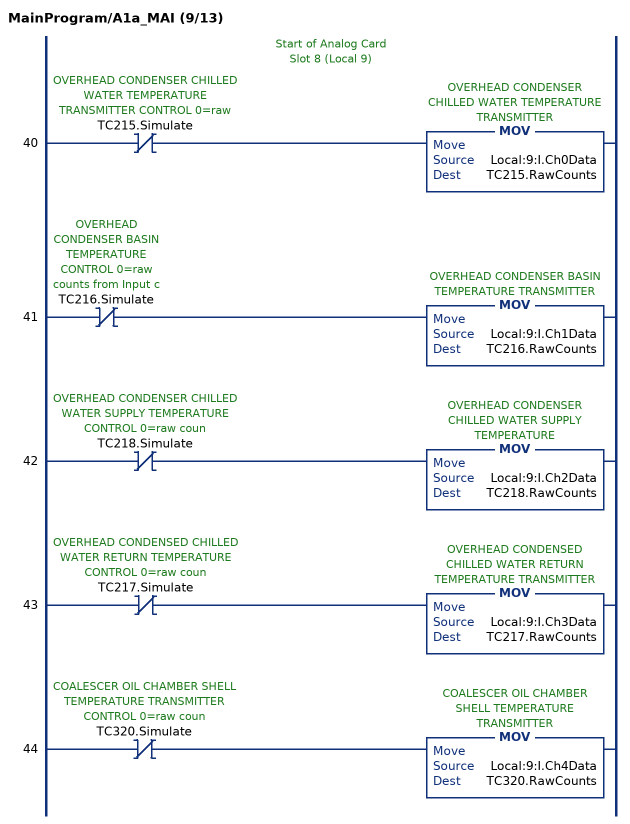
   // Start of Analog Card
   // Slot 8 (Local 9)
   40: XIO(TC215.Simulate)MOV(Local:9:I.Ch0Data,TC215.RawCounts);
   41: XIO(TC216.Simulate)MOV(Local:9:I.Ch1Data,TC216.RawCounts);
   42: XIO(TC218.Simulate)MOV(Local:9:I.Ch2Data,TC218.RawCounts);
   43: XIO(TC217.Simulate)MOV(Local:9:I.Ch3Data,TC217.RawCounts);
   44: XIO(TC320.Simulate)MOV(Local:9:I.Ch4Data,TC320.RawCounts);
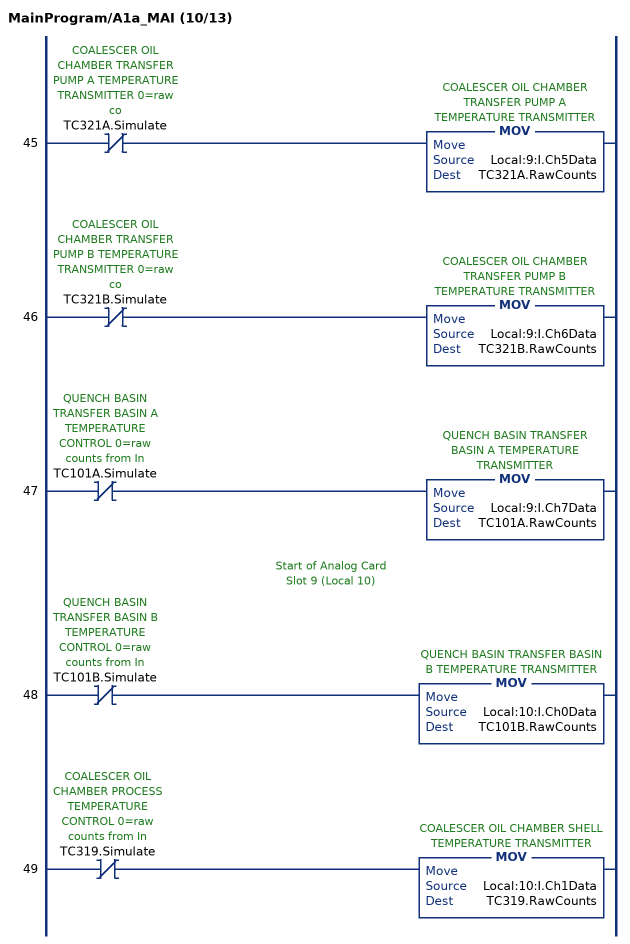
   45: XIO(TC321A.Simulate)MOV(Local:9:I.Ch5Data,TC321A.RawCounts);
   46: XIO(TC321B.Simulate)MOV(Local:9:I.Ch6Data,TC321B.RawCounts);
   47: XIO(TC101A.Simulate)MOV(Local:9:I.Ch7Data,TC101A.RawCounts);
   // Start of Analog Card
   // Slot 9 (Local 10)
   48: XIO(TC101B.Simulate)MOV(Local:10:I.Ch0Data,TC101B.RawCounts);
   49: XIO(TC319.Simulate)MOV(Local:10:I.Ch1Data,TC319.RawCounts);
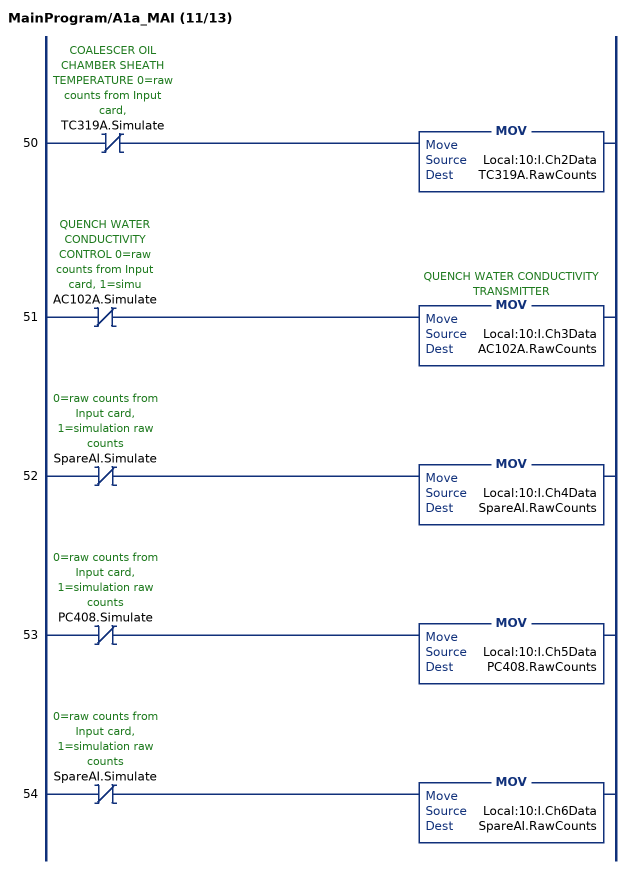
   50: XIO(TC319A.Simulate)MOV(Local:10:I.Ch2Data,TC319A.RawCounts);
   51: XIO(AC102A.Simulate)MOV(Local:10:I.Ch3Data,AC102A.RawCounts);
   52: XIO(SpareAI.Simulate)MOV(Local:10:I.Ch4Data,SpareAI.RawCounts);
   53: XIO(PC408.Simulate)MOV(Local:10:I.Ch5Data,PC408.RawCounts);
   54: XIO(SpareAI.Simulate)MOV(Local:10:I.Ch6Data,SpareAI.RawCounts);
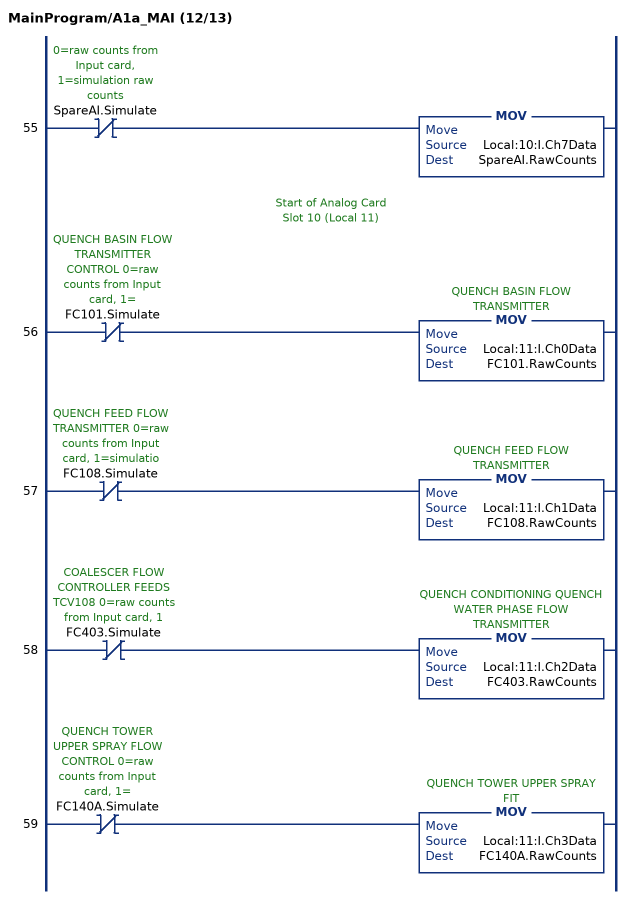
   55: XIO(SpareAI.Simulate)MOV(Local:10:I.Ch7Data,SpareAI.RawCounts);
   // Start of Analog Card
   // Slot 10 (Local 11)
   56: XIO(FC101.Simulate)MOV(Local:11:I.Ch0Data,FC101.RawCounts);
   57: XIO(FC108.Simulate)MOV(Local:11:I.Ch1Data,FC108.RawCounts);
   58: XIO(FC403.Simulate)MOV(Local:11:I.Ch2Data,FC403.RawCounts);
   59: XIO(FC140A.Simulate)MOV(Local:11:I.Ch3Data,FC140A.RawCounts);
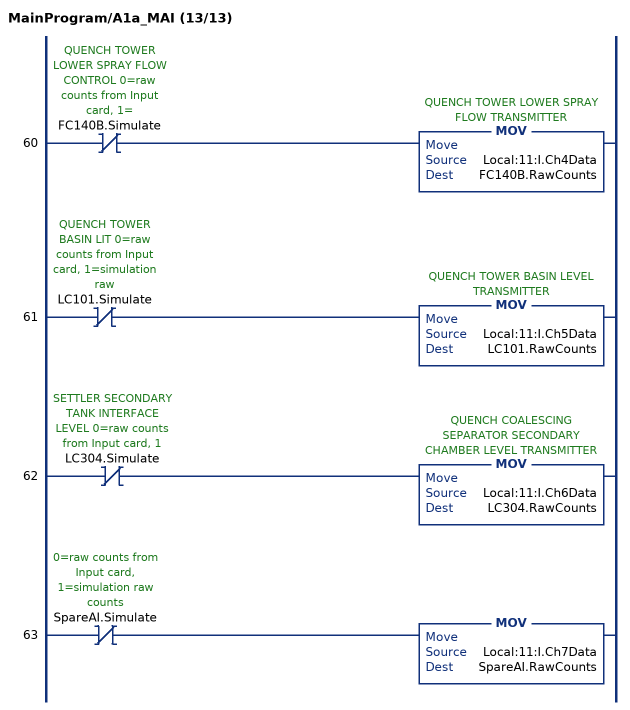
   60: XIO(FC140B.Simulate)MOV(Local:11:I.Ch4Data,FC140B.RawCounts);
   61: XIO(LC101.Simulate)MOV(Local:11:I.Ch5Data,LC101.RawCounts);
   62: XIO(LC304.Simulate)MOV(Local:11:I.Ch6Data,LC304.RawCounts);
   63: XIO(SpareAI.Simulate)MOV(Local:11:I.Ch7Data,SpareAI.RawCounts);
END_ROUTINE
